// TIA Portal project "HEAT-1-CADIZ-S71500_V9" (V20)

(* hardware
DEVICE "S7-1500/ET200MP station_1"  S7-1500 station
   slot 0: "Rail_0"  Rack  6ES7 590-1***0-0AA0
   slot 1: "PLC_1"  CPU 1517F-3 PN/DP  6ES7 517-3FP00-0AB0  V3.0
      slot 3: "CPU display_1"  6ES7591-1BA00-0AA0
      slot 32768: "PROFINET interface_1"  X1
         slot 32769: "Port_1"  X1 P1
         slot 32770: "Port_2"  X1 P2
      slot 33024: "PROFINET interface_2"  X2
         slot 33025: "Port_1"  X2 P1
      slot 33280: "DP interface_1"  X3
      slot 34817: "Virtual CP interface port_1"  Virtual CP interface port  Virtual CP interface port
DEVICE "GSD device_1"  GSD.Device.PN
   slot 0: "Rack"  Rack  V1.0
   slot 0: "KRC5"  KUKA.PROFINET 6.0  0x300  V6.0
      slot 0: "KUKA.PROFINET 6.0"  KUKA.PROFINET 6.0
      slot 1: "Interface1"  Interface1
         slot 1: "Port001(XF3)"  Port001(XF3)
         slot 2: "Port002(XF4)"  Port002(XF4)
         slot 3: "Port003(XF5)"  Port003(XF5)
         slot 4: "Port004(XF6)"  Port004(XF6)
   slot 1: "64 safe digital in- and outputs (2.4)_1"  64 safe digital in- and outputs (2.4)  KUKADevF64_2.4
      slot 0: "64 safe digital in- and outputs (2.4)"  64 safe digital in- and outputs (2.4)
   slot 2: "256 digital in- and outputs_1"  256 digital in- and outputs  KUKA Device IO256
      slot 0: "256 digital in- and outputs"  256 digital in- and outputs
DEVICE "ET 200SP station_2"  ET 200SP-Station
   slot 0: "Rack_0"  Rack  6ES5 710-8MAx1
   slot 0: "islaparking"  IM 155-6 PN ST  6ES7 155-6AU01-0BN0  V4.2
   slot 1: "DI 16x24VDC ST_1"  DI 16x24VDC ST  6ES7 131-6BH01-0BA0  V0.0
      slot 1: "DI 16x24VDC ST_1"  DI 16x24VDC ST
   slot 2: "DI 8x24VDC ST_1"  DI 8x24VDC ST  6ES7 131-6BF01-0BA0  V0.0
      slot 1: "DI 8x24VDC ST_1"  DI 8x24VDC ST
   slot 3: "DQ 16x24VDC/0.5A ST_1"  DQ 16x24VDC/0.5A ST  6ES7 132-6BH01-0BA0  V0.0
      slot 1: "DQ 16x24VDC/0.5A ST_1"  DQ 16x24VDC/0.5A ST
   slot 4: "DQ 8x24VDC/0.5A ST_1"  DQ 8x24VDC/0.5A ST  6ES7 132-6BF01-0BA0  V0.0
      slot 1: "DQ 8x24VDC/0.5A ST_1"  DQ 8x24VDC/0.5A ST
   slot 5: "Server module_1"  Server module  6ES7 193-6PA00-0AA0  V1.1
      slot 1: "Server module_1"  Server module
   slot 127: "BA 2xRJ45"  BA 2xRJ45  6ES7 193-6AR00-0AA0  V0.0
      slot 1: "Port_1"  X1 P1R  6ES7 193-6AR00-0AA0  V0.0
      slot 2: "Port_2"  X1 P2R  6ES7 193-6AR00-0AA0  V0.0
DEVICE "ET 200SP station_1"  ET 200SP-Station
   slot 0: "Rack_0"  Rack  6ES5 710-8MAx1
   slot 0: "islarobot"  IM 155-6 PN ST  6ES7 155-6AU01-0BN0  V4.2
   slot 1: "DI 16x24VDC ST_1"  DI 16x24VDC ST  6ES7 131-6BH01-0BA0  V0.0
      slot 1: "DI 16x24VDC ST_1"  DI 16x24VDC ST
   slot 2: "DI 8x24VDC ST_1"  DI 8x24VDC ST  6ES7 131-6BF01-0BA0  V0.0
      slot 1: "DI 8x24VDC ST_1"  DI 8x24VDC ST
   slot 3: "DQ 16x24VDC/0.5A ST_1"  DQ 16x24VDC/0.5A ST  6ES7 132-6BH01-0BA0  V0.0
      slot 1: "DQ 16x24VDC/0.5A ST_1"  DQ 16x24VDC/0.5A ST
   slot 4: "DQ 8x24VDC/0.5A ST_1"  DQ 8x24VDC/0.5A ST  6ES7 132-6BF01-0BA0  V0.0
      slot 1: "DQ 8x24VDC/0.5A ST_1"  DQ 8x24VDC/0.5A ST
   slot 5: "Server module_1"  Server module  6ES7 193-6PA00-0AA0  V1.1
      slot 1: "Server module_1"  Server module
   slot 127: "BA 2xRJ45"  BA 2xRJ45  6ES7 193-6AR00-0AA0  V0.0
      slot 1: "Port_1"  X1 P1R  6ES7 193-6AR00-0AA0  V0.0
      slot 2: "Port_2"  X1 P2R  6ES7 193-6AR00-0AA0  V0.0
*)

// ===== PLC "PLC_1"  CPU 1517F-3 PN/DP =====

VAR_GLOBAL   // PLC tag table "Default tag table"
   "RES1 (reservado)" AT %Q500.0 : Bool;
   "eStopButtonCabinet" AT %I40.0 : Bool;   // Emergency-Stop cabinet — 1oo2 result
   "eStopButtonTank" AT %I40.1 : Bool;   // Emergency-Stop tank — 1oo2 result
   "eStopButtonTankPartnerCh" AT %I41.1 : Bool;   // partner channel 1oo2 — do not use
   "eStopButtonWaterSystem" AT %I40.2 : Bool;   // Emergency-Stop water system — 1oo2 result
   "eStopButtonWaterSystemPartnerCh" AT %I41.2 : Bool;   // partner channel 1oo2 — do not use
   "eStopButtonHmiPanel" AT %I40.3 : Bool;   // Emergency-Stop HMI panel — 1oo2 result
   "eStopButtonHmiPanelPartnerCh" AT %I41.3 : Bool;   // partner channel 1oo2 — do not use
   "eStopButtonLightCurtain1" AT %I40.4 : Bool;   // Emergency-Stop light curtain 1 — 1oo2 resul
   "eStopButtonLightCurtain1PartnerCh" AT %I41.4 : Bool;   // partner channel 1oo2 — do not use
   "eStopButtonDoor" AT %I40.5 : Bool;   // Emergency-Stop Door — 1oo2 result
   "eStopButtonDoorPartnerCh" AT %I41.5 : Bool;   // partner channel 1oo2 — do not use
   "lightCurtain1Ossd1" AT %I50.0 : Bool;   // Z2 – LC 1 OSSD 1 (receiver)
   "lightCurtain1Ossd2" AT %I51.0 : Bool;   // Z2 – LC 1 OSSD 2 (receiver)
   "lightCurtain3Ossd1" AT %I50.1 : Bool;   // Z2 – LC 3 OSSD 1 (receiver)
   "lightCurtain3Ossd2" AT %I51.1 : Bool;   // Z2 – LC 3 OSSD 2 (receiver)
   "lightCurtain6Ossd1" AT %I50.2 : Bool;   // Z2 – LC 6 OSSD 1 (receiver)
   "lightCurtain6Ossd2" AT %I51.2 : Bool;   // Z2 – LC 6 OSSD 2 (receiver)
   "enableAccessReqSelector" AT %I50.3 : Bool;   // Rotary selector – enabless request access
   "DoorClosedCh1" AT %I50.6 : Bool;   // Safety door closed interlock – contact 1
   "resetDoorButton" AT %I50.7 : Bool;   // Reset push‑button
   "SAF_DOOR_CLSD_CH2" AT %I51.6 : Bool;   // Safety door closed interlock – contact 2
   "SAF_DOOR_UNLOCK_CH1" AT %Q60.0 : Bool;   // Unlock safety door – redundant output 1
   "SAF_GATE_UNLOCK_CH2" AT %Q60.2 : Bool;   // Unlock safety door – redundant output 2
   "IND_RESET_LAMP" AT %Q10.0 : Bool;   // Reset indicator lamp
   "IND_STATUS_LAMP" AT %Q10.1 : Bool;   // System-status pilot light
   "CMD_PRESS_EXH_VALVE" AT %Q11.0 : Bool;   // Pressure/exhaust solenoid-valve command
   "STS_RECIRC_PUMP" AT %I20.0 : Bool;   // Recirculation-pump feedback
   "STS_TRANSFER_PUMP" AT %I20.1 : Bool;   // Transfer-pump feedback
   "ALM_UV_FILTER" AT %I20.2 : Bool;   // UV-filter fault alarm
   "ALM_PIT_LVL_LOW" AT %I20.3 : Bool;   // Sump low-level alarm
   "ALM_TANK_LVL_LOW" AT %I20.4 : Bool;   // Tank low-level alarm
   "STS_TANK_FILLING" AT %I20.5 : Bool;   // Tank filling status
   "STS_TANK_DRAINING" AT %I20.6 : Bool;   // Tank draining status
   "CMD_TANK_FILL" AT %Q30.0 : Bool;   // Fill tank command
   "CMD_TANK_DRAIN" AT %Q30.1 : Bool;   // Drain tank command
   "MODE_WATER_MAN" AT %Q30.2 : Bool;   // Water system manual mode
   "MODE_WATER_AUTO" AT %Q30.3 : Bool;   // Water system automatic mode
   "IND_BEACON2_GREEN" AT %Q30.4 : Bool;   // Beacon 2 – green
   "IND_BEACON2_RED" AT %Q30.5 : Bool;   // Beacon 2 – red
   "robotPresenceSignalZone1" AT %I500.0 : Bool;
   "robotPresenceSignalZone2" AT %I500.1 : Bool;
   "robotPresenceSignalZone3" AT %I500.2 : Bool;
   "eStopButtonCabinetPartnerCh" AT %I41.0 : Bool;   // partner channel 1oo2 — do not use
   "lightCurtain2Ossd1" AT %I300.0 : Bool;
   "lightCurtain2Ossd2" AT %I301.0 : Bool;
   "eStopButtonIslandRightPartner" AT %I301.1 : Bool;
   "lightCurtain4Ossd1" AT %I350.0 : Bool;
   "eStopButtonIslandLeft" AT %I350.1 : Bool;
   "lightCurtain5Ossd1" AT %I350.2 : Bool;
   "eStopButtonIslandLefttPartner" AT %I350.3 : Bool;   // partner channel 1oo2 — do not use
   "lightCurtain4Ossd2" AT %I350.4 : Bool;
   "lightCurtain5Ossd2" AT %I350.6 : Bool;
   "accessReqButtonZone2" AT %I51.4 : Bool;   // Illuminated push-button – access request for zone 2
   "accessReqButtonZone3" AT %I51.5 : Bool;   // Illuminated push-button – access request for zone 3
   "accessReqButtonZone1" AT %I51.3 : Bool;   // Illuminated push-button – access request for zone 1
   "eStopButtonIslandRight" AT %I300.1 : Bool;
   "NHE – E‑Stop externo  NO pulsado" AT %Q500.1 : Bool;
   "BS – Puerta cerrada" AT %Q500.2 : Bool;
   "QBS – Ack puerta" AT %Q500.3 : Bool;
   "SHS1 – Stop 1" AT %Q500.4 : Bool;
   "SHS2 – Stop 2" AT %Q500.5 : Bool;
   "RES6" AT %Q500.6 : Bool;
   "RES7" AT %Q500.7 : Bool;
   "US2 – 24 V US2" AT %Q501.0 : Bool;
   "SBH – Safe Op Stop" AT %Q501.1 : Bool;
   "RES11" AT %Q501.2 : Bool;
   "RES12" AT %Q501.3 : Bool;
   "RES13" AT %Q501.4 : Bool;
   "RES14" AT %Q501.5 : Bool;
   "RES15" AT %Q501.6 : Bool;
   "SPA – Power‑down Ack" AT %Q501.7 : Bool;
   "resetHmiButton" AT %I51.7 : Bool;
   "Tag_1" AT %M200.0 : Bool;
   "Tag_2" AT %M201.0 : Bool;
   "Tag_3" AT %M500.1 : Bool;
   "Tag_4" AT %M755.5 : Bool;
   "Tag_5" AT %QB600 : Byte;
   "V5" AT %Q0.4 : Bool;
   "ABRIR_TAPA_PEPA" AT %Q170.2 : Bool;
   "CERRAR_TAPA_PEPA" AT %Q170.3 : Bool;
   "ABRIR_TAPA_INMERSION" AT %Q170.4 : Bool;
   "CERRAR_TAPA_INMERSION" AT %Q170.5 : Bool;
   "ABRIR_TAPA_MARCADOR" AT %Q170.6 : Bool;
   "CERRAR_TAPA_MARCADOR" AT %Q170.7 : Bool;
   "ABRIR_TAPA_PERFILOMETRO" AT %Q171.0 : Bool;
   "CERRAR_TAPA_PERFILOMETRO" AT %Q171.1 : Bool;
   "V6" AT %Q0.5 : Bool;
   "V7" AT %Q0.6 : Bool;
   "V8" AT %Q0.7 : Bool;
END_VAR

VAR_GLOBAL   // PLC tag table "Robot Jog"
   "tcpTargetX_01" AT %Q600.1 : Bool;
   "tcpTargetX_02" AT %Q600.2 : Bool;
   "tcpTargetX_03" AT %Q600.3 : Bool;
   "tcpTargetX_04" AT %Q600.4 : Bool;
   "tcpTargetX_05" AT %Q600.5 : Bool;
   "tcpTargetX_08" AT %Q601.0 : Bool;
   "tcpTargetX_16" AT %Q602.0 : Bool;
   "tcpTargetX_17" AT %Q602.1 : Bool;
   "tcpTargetX_06" AT %Q600.6 : Bool;
   "tcpTargetX_07" AT %Q600.7 : Bool;
   "tcpTargetX_09" AT %Q601.1 : Bool;
   "tcpTargetX_10" AT %Q601.2 : Bool;
   "tcpTargetX_11" AT %Q601.3 : Bool;
   "tcpTargetX_12" AT %Q601.4 : Bool;
   "tcpTargetX_13" AT %Q601.5 : Bool;
   "tcpTargetX_14" AT %Q601.6 : Bool;
   "tcpTargetX_15" AT %Q601.7 : Bool;
   "tcpTargetX_18" AT %Q602.2 : Bool;
   "tcpTargetX_19" AT %Q602.3 : Bool;
   "tcpTargetX_20" AT %Q602.4 : Bool;
   "tcpTargetX_21" AT %Q602.5 : Bool;
   "tcpTargetX_22" AT %Q602.6 : Bool;
   "tcpTargetX_23" AT %Q602.7 : Bool;
   "tcpTargetX_24" AT %Q603.0 : Bool;
   "tcpTargetX_25" AT %Q603.1 : Bool;
   "tcpTargetX_26" AT %Q603.2 : Bool;
   "tcpTargetX_27" AT %Q603.3 : Bool;
   "tcpTargetX_28" AT %Q603.4 : Bool;
   "tcpTargetX_29" AT %Q603.5 : Bool;
   "tcpTargetX_30" AT %Q603.6 : Bool;
   "tcpTargetX_31" AT %Q603.7 : Bool;
   "tcpTargetY_00" AT %Q604.0 : Bool;
   "tcpTargetY_01" AT %Q604.1 : Bool;
   "tcpTargetY_02" AT %Q604.2 : Bool;
   "tcpTargetY_03" AT %Q604.3 : Bool;
   "tcpTargetY_04" AT %Q604.4 : Bool;
   "tcpTargetY_05" AT %Q604.5 : Bool;
   "tcpTargetY_06" AT %Q604.6 : Bool;
   "tcpTargetY_07" AT %Q604.7 : Bool;
   "tcpTargetY_08" AT %Q605.0 : Bool;
   "tcpTargetY_09" AT %Q605.1 : Bool;
   "tcpTargetY_10" AT %Q605.2 : Bool;
   "tcpTargetY_11" AT %Q605.3 : Bool;
   "tcpTargetY_12" AT %Q605.4 : Bool;
   "tcpTargetY_13" AT %Q605.5 : Bool;
   "tcpTargetY_14" AT %Q605.6 : Bool;
   "tcpTargetY_15" AT %Q605.7 : Bool;
   "tcpTargetY_16" AT %Q606.0 : Bool;   // $IN[49]
   "tcpTargetY_17" AT %Q606.1 : Bool;   // $IN[50]
   "tcpTargetY_18" AT %Q606.2 : Bool;   // $IN[51]
   "tcpTargetY_19" AT %Q606.3 : Bool;   // true
   "tcpTargetY_20" AT %Q606.4 : Bool;
   "tcpTargetY_21" AT %Q606.5 : Bool;   // true
   "tcpTargetY_22" AT %Q606.6 : Bool;   // true
   "tcpTargetY_23" AT %Q606.7 : Bool;   // true
   "tcpTargetY_24" AT %Q607.0 : Bool;   // true
   "tcpTargetY_25" AT %Q607.1 : Bool;   // true
   "tcpTargetY_26" AT %Q607.2 : Bool;   // true
   "tcpTargetY_27" AT %Q607.3 : Bool;
   "tcpTargetY_28" AT %Q607.4 : Bool;
   "tcpTargetY_29" AT %Q607.5 : Bool;
   "tcpTargetY_30" AT %Q607.6 : Bool;
   "tcpTargetY_31" AT %Q607.7 : Bool;
   "tcpTargetZ_00" AT %Q608.0 : Bool;
   "tcpTargetZ_01" AT %Q608.1 : Bool;
   "tcpTargetZ_02" AT %Q608.2 : Bool;
   "tcpTargetZ_03" AT %Q608.3 : Bool;
   "tcpTargetZ_04" AT %Q608.4 : Bool;
   "tcpTargetZ_05" AT %Q608.5 : Bool;
   "tcpTargetZ_06" AT %Q608.6 : Bool;
   "tcpTargetZ_07" AT %Q608.7 : Bool;
   "tcpTargetZ_08" AT %Q609.0 : Bool;
   "tcpTargetZ_09" AT %Q609.1 : Bool;
   "tcpTargetZ_10" AT %Q609.2 : Bool;
   "tcpTargetZ_11" AT %Q609.3 : Bool;
   "tcpTargetZ_12" AT %Q609.4 : Bool;
   "tcpTargetZ_13" AT %Q609.5 : Bool;
   "tcpTargetZ_14" AT %Q609.6 : Bool;
   "tcpTargetZ_15" AT %Q609.7 : Bool;
   "tcpTargetZ_16" AT %Q610.0 : Bool;
   "tcpTargetZ_17" AT %Q610.1 : Bool;
   "tcpTargetZ_18" AT %Q610.2 : Bool;
   "tcpTargetZ_19" AT %Q610.3 : Bool;
   "tcpTargetZ_20" AT %Q610.4 : Bool;
   "tcpTargetZ_21" AT %Q610.5 : Bool;
   "tcpTargetZ_22" AT %Q610.6 : Bool;
   "tcpTargetZ_23" AT %Q610.7 : Bool;
   "tcpTargetZ_24" AT %Q611.0 : Bool;
   "tcpTargetZ_25" AT %Q611.1 : Bool;
   "tcpTargetZ_26" AT %Q611.2 : Bool;
   "tcpTargetZ_27" AT %Q611.3 : Bool;
   "tcpTargetZ_28" AT %Q611.4 : Bool;
   "tcpTargetZ_29" AT %Q611.5 : Bool;
   "tcpTargetZ_30" AT %Q611.6 : Bool;
   "tcpTargetZ_31" AT %Q611.7 : Bool;
   "e1Target_00" AT %Q612.0 : Bool;
   "e1Target_01" AT %Q612.1 : Bool;
   "e1Target_02" AT %Q612.2 : Bool;
   "e1Target_03" AT %Q612.3 : Bool;
   "e1Target_04" AT %Q612.4 : Bool;
   "e1Target_05" AT %Q612.5 : Bool;
   "e1Target_06" AT %Q612.6 : Bool;
   "e1Target_07" AT %Q612.7 : Bool;
   "e1Target_08" AT %Q613.0 : Bool;
   "e1Target_09" AT %Q613.1 : Bool;
   "e1Target_10" AT %Q613.2 : Bool;
   "e1Target_11" AT %Q613.3 : Bool;
   "e1Target_12" AT %Q613.4 : Bool;
   "e1Target_13" AT %Q613.5 : Bool;
   "e1Target_14" AT %Q613.6 : Bool;
   "e1Target_15" AT %Q613.7 : Bool;
   "e1Target_16" AT %Q614.0 : Bool;
   "e1Target_17" AT %Q614.1 : Bool;
   "e1Target_18" AT %Q614.2 : Bool;
   "e1Target_19" AT %Q614.3 : Bool;
   "e1Target_20" AT %Q614.4 : Bool;
   "e1Target_21" AT %Q614.5 : Bool;
   "e1Target_22" AT %Q614.6 : Bool;
   "e1Target_23" AT %Q614.7 : Bool;
   "e1Target_24" AT %Q615.0 : Bool;
   "e1Target_25" AT %Q615.1 : Bool;
   "e1Target_26" AT %Q615.2 : Bool;
   "e1Target_27" AT %Q615.3 : Bool;
   "e1Target_28" AT %Q615.4 : Bool;
   "e1Target_29" AT %Q615.5 : Bool;
   "e1Target_30" AT %Q615.6 : Bool;
   "e1Target_31" AT %Q615.7 : Bool;
   "e1Target_Word" AT %QD612 : DWord;
   "moveCodeKuka" AT %QW616 : Word;   // SIGNAL goTrrigger $IN[ 129]
   "rbDone" AT %I624.0 : Bool;   // SIGNAL rbDoneEdge $OUT[193]
   "x1Target_Word" AT %QD600 : DWord;
   "y1Target_Word" AT %QD604 : DWord;
   "z1Target_Word" AT %QD608 : DWord;
   "goTrigger" AT %Q618.0 : Bool;
END_VAR

VAR_GLOBAL   // PLC tag table "Robot Position"
   "tcpPosX_00" AT %I600.0 : Bool;
   "tcpPosX_01" AT %I600.1 : Bool;
   "tcpPosX_02" AT %I600.2 : Bool;
   "tcpPosX_03" AT %I600.3 : Bool;
   "tcpPosX_04" AT %I600.4 : Bool;
   "tcpPosX_05" AT %I600.5 : Bool;
   "tcpPosX_06" AT %I600.6 : Bool;
   "tcpPosX_07" AT %I600.7 : Bool;
   "tcpPosX_08" AT %I601.0 : Bool;
   "tcpPosX_09" AT %I601.1 : Bool;
   "tcpPosX_10" AT %I601.2 : Bool;
   "tcpPosX_11" AT %I601.3 : Bool;
   "tcpPosX_12" AT %I601.4 : Bool;
   "tcpPosX_13" AT %I601.5 : Bool;
   "tcpPosX_14" AT %I601.6 : Bool;
   "tcpPosX_15" AT %I601.7 : Bool;
   "tcpPosX_16" AT %I602.0 : Bool;
   "tcpPosX_17" AT %I602.1 : Bool;
   "tcpPosX_18" AT %I602.2 : Bool;
   "tcpPosX_19" AT %I602.3 : Bool;
   "tcpPosX_20" AT %I602.4 : Bool;
   "tcpPosX_21" AT %I602.5 : Bool;
   "tcpPosX_22" AT %I602.6 : Bool;
   "tcpPosX_23" AT %I602.7 : Bool;
   "tcpPosX_24" AT %I603.0 : Bool;
   "tcpPosX_25" AT %I603.1 : Bool;
   "tcpPosX_26" AT %I603.2 : Bool;
   "tcpPosX_27" AT %I603.3 : Bool;
   "tcpPosX_28" AT %I603.4 : Bool;
   "tcpPosX_29" AT %I603.5 : Bool;
   "tcpPosX_30" AT %I603.6 : Bool;
   "tcpPosX_31" AT %I603.7 : Bool;
   "tcpPosY_00" AT %I604.0 : Bool;
   "tcpPosY_01" AT %I604.1 : Bool;
   "tcpPosY_02" AT %I604.2 : Bool;
   "tcpPosY_03" AT %I604.3 : Bool;
   "tcpPosY_04" AT %I604.4 : Bool;
   "tcpPosY_05" AT %I604.5 : Bool;
   "tcpPosY_06" AT %I604.6 : Bool;
   "tcpPosY_07" AT %I604.7 : Bool;
   "tcpPosY_08" AT %I605.0 : Bool;
   "tcpPosY_09" AT %I605.1 : Bool;
   "tcpPosY_10" AT %I605.2 : Bool;
   "tcpPosY_11" AT %I605.3 : Bool;
   "tcpPosY_12" AT %I605.4 : Bool;
   "tcpPosY_13" AT %I605.5 : Bool;
   "tcpPosY_14" AT %I605.6 : Bool;
   "tcpPosY_15" AT %I605.7 : Bool;
   "tcpPosY_16" AT %I606.0 : Bool;
   "tcpPosY_17" AT %I606.1 : Bool;
   "tcpPosY_18" AT %I606.2 : Bool;
   "tcpPosY_19" AT %I606.3 : Bool;
   "tcpPosY_20" AT %I606.4 : Bool;
   "tcpPosY_21" AT %I606.5 : Bool;
   "tcpPosY_22" AT %I606.6 : Bool;
   "tcpPosY_23" AT %I606.7 : Bool;
   "tcpPosY_24" AT %I607.0 : Bool;
   "tcpPosY_25" AT %I607.1 : Bool;
   "tcpPosY_26" AT %I607.2 : Bool;
   "tcpPosY_27" AT %I607.3 : Bool;
   "tcpPosY_28" AT %I607.4 : Bool;
   "tcpPosY_29" AT %I607.5 : Bool;
   "tcpPosY_30" AT %I607.6 : Bool;
   "tcpPosY_31" AT %I607.7 : Bool;
   "tcpPosZ_00" AT %I608.0 : Bool;
   "tcpPosZ_01" AT %I608.1 : Bool;
   "tcpPosZ_02" AT %I608.2 : Bool;
   "tcpPosZ_03" AT %I608.3 : Bool;
   "tcpPosZ_04" AT %I608.4 : Bool;
   "tcpPosZ_05" AT %I608.5 : Bool;
   "tcpPosZ_06" AT %I608.6 : Bool;
   "tcpPosZ_07" AT %I608.7 : Bool;
   "tcpPosZ_08" AT %I609.0 : Bool;
   "tcpPosZ_09" AT %I609.1 : Bool;
   "tcpPosZ_10" AT %I609.2 : Bool;
   "tcpPosZ_11" AT %I609.3 : Bool;
   "tcpPosZ_12" AT %I609.4 : Bool;
   "tcpPosZ_13" AT %I609.5 : Bool;
   "tcpPosZ_14" AT %I609.6 : Bool;
   "tcpPosZ_15" AT %I609.7 : Bool;
   "tcpPosZ_16" AT %I610.0 : Bool;
   "tcpPosZ_17" AT %I610.1 : Bool;
   "tcpPosZ_18" AT %I610.2 : Bool;
   "tcpPosZ_19" AT %I610.3 : Bool;
   "tcpPosZ_20" AT %I610.4 : Bool;
   "tcpPosZ_21" AT %I610.5 : Bool;
   "tcpPosZ_22" AT %I610.6 : Bool;
   "tcpPosZ_23" AT %I610.7 : Bool;
   "tcpPosZ_24" AT %I611.0 : Bool;
   "tcpPosZ_25" AT %I611.1 : Bool;
   "tcpPosZ_26" AT %I611.2 : Bool;
   "tcpPosZ_27" AT %I611.3 : Bool;
   "tcpPosZ_28" AT %I611.4 : Bool;
   "tcpPosZ_29" AT %I611.5 : Bool;
   "tcpPosZ_30" AT %I611.6 : Bool;
   "tcpPosZ_31" AT %I611.7 : Bool;
   "tcpPosA_00" AT %I612.0 : Bool;
   "tcpPosA_01" AT %I612.1 : Bool;
   "tcpPosA_02" AT %I612.2 : Bool;
   "tcpPosA_03" AT %I612.3 : Bool;
   "tcpPosA_04" AT %I612.4 : Bool;
   "tcpPosA_05" AT %I612.5 : Bool;
   "tcpPosA_06" AT %I612.6 : Bool;
   "tcpPosA_07" AT %I612.7 : Bool;
   "tcpPosA_08" AT %I613.0 : Bool;
   "tcpPosA_09" AT %I613.1 : Bool;
   "tcpPosA_10" AT %I613.2 : Bool;
   "tcpPosA_11" AT %I613.3 : Bool;
   "tcpPosA_12" AT %I613.4 : Bool;
   "tcpPosA_13" AT %I613.5 : Bool;
   "tcpPosA_14" AT %I613.6 : Bool;
   "tcpPosA_15" AT %I613.7 : Bool;
   "tcpPosA_16" AT %I614.0 : Bool;
   "tcpPosA_17" AT %I614.1 : Bool;
   "tcpPosA_18" AT %I614.2 : Bool;
   "tcpPosA_19" AT %I614.3 : Bool;
   "tcpPosA_20" AT %I614.4 : Bool;
   "tcpPosA_21" AT %I614.5 : Bool;
   "tcpPosA_22" AT %I614.6 : Bool;
   "tcpPosA_23" AT %I614.7 : Bool;
   "tcpPosA_24" AT %I615.0 : Bool;
   "tcpPosA_25" AT %I615.1 : Bool;
   "tcpPosA_26" AT %I615.2 : Bool;
   "tcpPosA_27" AT %I615.3 : Bool;
   "tcpPosA_28" AT %I615.4 : Bool;
   "tcpPosA_29" AT %I615.5 : Bool;
   "tcpPosA_30" AT %I615.6 : Bool;
   "tcpPosA_31" AT %I615.7 : Bool;
   "tcpPosB_00" AT %I616.0 : Bool;
   "tcpPosB_01" AT %I616.1 : Bool;
   "tcpPosB_02" AT %I616.2 : Bool;
   "tcpPosB_03" AT %I616.3 : Bool;
   "tcpPosB_04" AT %I616.4 : Bool;
   "tcpPosB_05" AT %I616.5 : Bool;
   "tcpPosB_06" AT %I616.6 : Bool;
   "tcpPosB_07" AT %I616.7 : Bool;
   "tcpPosB_08" AT %I617.0 : Bool;
   "tcpPosB_09" AT %I617.1 : Bool;
   "tcpPosB_10" AT %I617.2 : Bool;
   "tcpPosB_11" AT %I617.3 : Bool;
   "tcpPosB_12" AT %I617.4 : Bool;
   "tcpPosB_13" AT %I617.5 : Bool;
   "tcpPosB_14" AT %I617.6 : Bool;
   "tcpPosB_15" AT %I617.7 : Bool;
   "tcpPosB_16" AT %I618.0 : Bool;
   "tcpPosB_17" AT %I618.1 : Bool;
   "tcpPosB_18" AT %I618.2 : Bool;
   "tcpPosB_19" AT %I618.3 : Bool;
   "tcpPosB_20" AT %I618.4 : Bool;
   "tcpPosB_21" AT %I618.5 : Bool;
   "tcpPosB_22" AT %I618.6 : Bool;
   "tcpPosB_23" AT %I618.7 : Bool;
   "tcpPosB_24" AT %I619.0 : Bool;
   "tcpPosB_25" AT %I619.1 : Bool;
   "tcpPosB_26" AT %I619.2 : Bool;
   "tcpPosB_27" AT %I619.3 : Bool;
   "tcpPosB_28" AT %I619.4 : Bool;
   "tcpPosB_29" AT %I619.5 : Bool;
   "tcpPosB_30" AT %I619.6 : Bool;
   "tcpPosB_31" AT %I619.7 : Bool;
   "tcpPosC_00" AT %I620.0 : Bool;
   "tcpPosC_01" AT %I620.1 : Bool;
   "tcpPosC_02" AT %I620.2 : Bool;
   "tcpPosC_03" AT %I620.3 : Bool;
   "tcpPosC_04" AT %I620.4 : Bool;
   "tcpPosC_05" AT %I620.5 : Bool;
   "tcpPosC_06" AT %I620.6 : Bool;
   "tcpPosC_07" AT %I620.7 : Bool;
   "tcpPosC_08" AT %I621.0 : Bool;
   "tcpPosC_09" AT %I621.1 : Bool;
   "tcpPosC_10" AT %I621.2 : Bool;
   "tcpPosC_11" AT %I621.3 : Bool;
   "tcpPosC_12" AT %I621.4 : Bool;
   "tcpPosC_13" AT %I621.5 : Bool;
   "tcpPosC_14" AT %I621.6 : Bool;
   "tcpPosC_15" AT %I621.7 : Bool;
   "tcpPosC_16" AT %I622.0 : Bool;
   "tcpPosC_17" AT %I622.1 : Bool;
   "tcpPosC_18" AT %I622.2 : Bool;
   "tcpPosC_19" AT %I622.3 : Bool;
   "tcpPosC_20" AT %I622.4 : Bool;
   "tcpPosC_21" AT %I622.5 : Bool;
   "tcpPosC_22" AT %I622.6 : Bool;
   "tcpPosC_23" AT %I622.7 : Bool;
   "tcpPosC_24" AT %I623.0 : Bool;
   "tcpPosC_25" AT %I623.1 : Bool;
   "tcpPosC_26" AT %I623.2 : Bool;
   "tcpPosC_27" AT %I623.3 : Bool;
   "tcpPosC_28" AT %I623.4 : Bool;
   "tcpPosC_29" AT %I623.5 : Bool;
   "tcpPosC_30" AT %I623.6 : Bool;
   "tcpPosC_31" AT %I623.7 : Bool;
   "tcpPosE1_01" AT %I628.0 : Bool;
   "tcpPosE1_02" AT %I628.1 : Bool;
   "tcpPosE1_03" AT %I628.2 : Bool;
   "tcpPosE1_04" AT %I628.3 : Bool;
   "tcpPosE1_05" AT %I628.4 : Bool;
   "tcpPosE1_06" AT %I628.5 : Bool;
   "tcpPosE1_07" AT %I628.6 : Bool;
   "tcpPosE1_08" AT %I628.7 : Bool;
   "tcpPosE1_09" AT %I629.0 : Bool;
   "tcpPosE1_10" AT %I629.1 : Bool;
   "tcpPosE1_11" AT %I629.2 : Bool;
   "tcpPosE1_12" AT %I629.3 : Bool;
   "tcpPosE1_13" AT %I629.4 : Bool;
   "tcpPosE1_14" AT %I629.5 : Bool;
   "tcpPosE1_15" AT %I629.6 : Bool;
   "tcpPosE1_16" AT %I629.7 : Bool;
   "tcpPosE1_17" AT %I630.0 : Bool;
   "tcpPosE1_18" AT %I630.1 : Bool;
   "tcpPosE1_19" AT %I630.2 : Bool;
   "tcpPosE1_20" AT %I630.3 : Bool;
   "tcpPosE1_21" AT %I630.4 : Bool;
   "tcpPosE1_22" AT %I630.5 : Bool;
   "tcpPosE1_23" AT %I630.6 : Bool;
   "tcpPosE1_24" AT %I630.7 : Bool;
   "tcpPosE1_25" AT %I631.0 : Bool;
   "tcpPosE1_26" AT %I631.1 : Bool;
   "tcpPosE1_27" AT %I631.2 : Bool;
   "tcpPosE1_28" AT %I631.3 : Bool;
   "tcpPosE1_29" AT %I631.4 : Bool;
   "tcpPosE1_30" AT %I631.5 : Bool;
   "tcpPosE1_31" AT %I631.6 : Bool;
   "tcpPosE1_32" AT %I631.7 : Bool;
   "tcpX_rawLe32" AT %ID600 : DWord;
   "tcpY_rawLe32" AT %ID604 : DWord;
   "tcpZ_rawLe32" AT %ID608 : DWord;
   "tcpB_rawLe32" AT %ID616 : DWord;
   "tcpC_rawLe32" AT %ID620 : DWord;
   "e1_rawLe32" AT %ID628 : DWord;
   "tcpA_rawLe32" AT %ID612 : DWord;
END_VAR

VAR_GLOBAL   // PLC tag table "Tool Change"
   "dockSensorToolInPosition" AT %I150.0 : Bool;   // DETECTOR_YUGO_LP
   "dockSensorCoverClosed" AT %I150.1 : Bool;   // TAPA_CERRADA_YUGO_LP
   "dockSensorCoverOpen" AT %I160.0 : Bool;   // TAPA_ABIERTA_YUGO_LP
   "dockValveV2UnlockOn" AT %Q171.2 : Bool;   // SOLTAR_HERRAMIENTA_YUGO_LP / CAMBIA A FALSE
   "dockValveCoverOpenOn" AT %Q170.0 : Bool;   // ABRIR_TAPA_YUGO_LP
   "dockValveCoverCloseOn" AT %Q170.1 : Bool;   // CERRAR_TAPA_YUGO_LP
   "robotSensorMpsUnlocked" AT %I200.0 : Bool;   // INTERCAMBIO_DESBLOQUEADO_LR
   "robotSensorMpsLocked" AT %I200.1 : Bool;   // INTERCAMBIO_BLOQUEADO_LR
   "robotSensorMpsCoupled" AT %I200.2 : Bool;   // HERRAMIENTA_PUESTA_LR /AL COLOCAR METAL
   "robotSensorMpsCtrlAirPressureOk" AT %I200.3 : Bool;   // PRESION_CORRECTA_LR
   "kukaFeedbackDockToolInPosition" AT %Q618.1 : Bool;   // INKUKA_DETECTOR_HERRAMIENTA
   "kukaFeedbackDockCoverClosed" AT %Q618.2 : Bool;   // INKUKA_TAPA_CERRADA_YUGO
   "kukaFeedbackDockCoverOpen" AT %Q618.3 : Bool;   // INKUKA_TAPA_ABIERTA_YUGO
   "kukaFeedbackRobotMpsUnlocked" AT %Q618.4 : Bool;   // INKUKA_INTERCAMBIO_DESBLOQUEADO
   "kukaFeedbackRobotMpsLocked" AT %Q618.5 : Bool;   // INKUKA_INTERCAMBIO_BLOQUEADO
   "kukaFeedbackRobotMpsCoupled" AT %Q618.6 : Bool;   // INKUKA_HERRAMIENTA_PUESTA /AL COLOCAR util met
   "kukaFeedbackRobotMpsCtrlAirPressureOk" AT %Q618.7 : Bool;
   "kukaCmdUnlockMps" AT %I624.1 : Bool;   // OUTKUKA_SOLTAR_HERRAMIENTA_YUGO
   "kukaCmdOpenCover" AT %I624.2 : Bool;   // OUTKUKA_ABRIR_TAPA_YUGO
   "kukaCmdCloseCover" AT %I624.3 : Bool;   // OUTKUKA_CERRAR_TAPA_YUGO
   "V1_B14_S2" AT %Q0.0 : Bool;
   "V1_B12_S4" AT %Q0.1 : Bool;
   "V2_B14_S2" AT %Q0.2 : Bool;
   "V2_B12_S4" AT %Q0.3 : Bool;
END_VAR

// folder: 10. System/DbsInstancia

DATA_BLOCK "InstKukaControlSeq"   // DB14
{ S7_Optimized_Access := 'TRUE' }
VERSION : 0.1
// stored: InstanceOfName KukaControlSeq
"KukaControlSeq"
BEGIN
END_DATA_BLOCK

DATA_BLOCK "InstSupervisorSeq"   // DB15
{ S7_Optimized_Access := 'TRUE' }
VERSION : 0.1
// stored: InstanceOfName SupervisorSeq
"SupervisorSeq"
BEGIN
END_DATA_BLOCK

DATA_BLOCK "InstSeqManager"   // DB16
{ S7_Optimized_Access := 'TRUE' }
VERSION : 0.1
// stored: InstanceOfName SeqManager
"SeqManager"
BEGIN
END_DATA_BLOCK

// folder: 10. System/DbsOpcUa

DATA_BLOCK "PlcStatus"   // DB4
{ S7_Optimized_Access := 'TRUE' }
VERSION : 0.1
   VAR
      mode : Struct
         effective : UInt;
         ready : Bool;
      END_STRUCT;
      active : Struct
         baseId : UInt;
         toolId : UInt;
         profileId : UInt;
      END_STRUCT;
      exec : Struct
         ackSeq : UInt;
         accepted : Bool;
         busy : Bool;
         done : Bool;
         error : Bool;
         errorCode : UDInt;
      END_STRUCT;
      pose : Struct
         tcpPosX_mm : LReal;
         tcpPosY_mm : LReal;
         tcpPosZ_mm : LReal;
         tcpOriA_deg : LReal;
         tcpOriB_deg : LReal;
         tcpOriC_deg : LReal;
         e1Pos_mm : LReal;
      END_STRUCT;
      Supervisor : Struct
         global : Struct
            heartBeatPlc : Bool;
            stepPlc : Int;
            plcOk : Bool;
            safetyOk : Bool;
            airOk : Bool;
            inspWaterOk : Bool;
            tankWaterOk : Bool;
            robotOk : Bool;
            acknowledge : Bool;
         END_STRUCT;
         identification : Struct
            carriageId : UInt;
            newCarriageId : Bool;
            idRunning : Bool;
         END_STRUCT;
         startUs : Struct
            startUsReady : Bool;
         END_STRUCT;
         stopUs : Struct
            stopUsReady : Bool;
         END_STRUCT;
         "deadElementCheck&Balancing" : Struct
            paCheckReady : Bool;
         END_STRUCT;
         gaintAdjustment : Struct
            gainReady : Bool;
         END_STRUCT;
         "tcgCheck&Adj" : Struct
            tcgReady : Bool;
         END_STRUCT;
         scanGeneric : Struct
            idScan : String;
            pointOrigin : LReal;
            xSize : LReal;
            ySize : LReal;
         END_STRUCT;
         scanRefPart : Struct
            scanRefStart : Bool;
         END_STRUCT;
         scanInsPart : Struct
            scanInspStart : Bool;
         END_STRUCT;
         preEval : Struct
            markRunning : Bool;
            markState : Bool;
         END_STRUCT;
         "break/Unbreak" : Struct
            breakUs : Bool;
            unbreakUs : Bool;
         END_STRUCT;
         rescanning : Struct
            robotRescanning : Bool;
         END_STRUCT;
         error : Struct
            acknowledgeError : Bool;
         END_STRUCT;
      END_STRUCT;
   END_VAR
BEGIN
END_DATA_BLOCK

DATA_BLOCK "KukaControlCmd"   // DB5
{ S7_Optimized_Access := 'TRUE' }
VERSION : 0.1
   VAR
      code : UInt;
      seq : UInt;
      tcpTargetX_mm : LReal;
      tcpTargetY_mm : LReal;
      tcpTargetZ_mm : LReal;
      e1Target : LReal;
      toolRequestId : UInt;
      baseRequestId : UInt;
      profileRequestId : UInt;
      vel_mms : LReal;
      index_mm : LReal;
      apo_mm : LReal;
      mode : Struct
         request : UInt;
         reqSeq : UInt;
      END_STRUCT;
   END_VAR
BEGIN
END_DATA_BLOCK

DATA_BLOCK "SupervisorCmd"   // DB6
{ S7_Optimized_Access := 'TRUE' }
VERSION : 0.1
   VAR
      global : Struct
         heartBeatSupervisor : Bool;
         stepSupervisor : Int;
         supervisorOk : Bool;
         stateUs : Bool;
      END_STRUCT;
      request : Struct
         reqCarriageId : Bool;
         reqRefPart : Bool;
         reqStopCycle : Bool;
         reqTcgAdj : Bool;
         reqId : Bool;
         reqPreEval : Bool;
         reqIdentificationState : Bool;
         reqMark : Bool;
      END_STRUCT;
      identification : Struct
         pns : String;
         referencePart : String;
         endEffector : Int;
         utTech : UInt;
         teachReq : Bool;
         paCheckReq : Bool;
         tcgReq : Bool;
      END_STRUCT;
      startUs : Struct
         startUsRunning : Bool;
      END_STRUCT;
      stopUs : Struct
         stopUsRunning : Bool;
      END_STRUCT;
      "deadElementCheck&Balancing" : Struct
         elemState : Bool;
         elemRunning : Bool;
         balState : Bool;
         balRunning : Bool;
      END_STRUCT;
      gainAdjustment : Struct
         gainState : Bool;
         gainRunning : Bool;
      END_STRUCT;
      "tcgCheck&Adj" : Struct
         tcgInProgress : Bool;
         tcgNextStep : Bool;
         tcgState : Bool;
      END_STRUCT;
      scanRefPart : Struct
         scanRefState : Bool;
         scanRefRunning : Bool;
      END_STRUCT;
      scanInspPart : Struct
         scanInspState : Bool;
         scanInspRunning : Bool;
      END_STRUCT;
      preEval : Struct
         pointCoordinates : LReal;
      END_STRUCT;
      rescanning : Struct
         goBack : Bool;
         rescanning : Bool;
      END_STRUCT;
      error : Struct
         errorMessage : String;
         errorOcurred : Bool;
      END_STRUCT;
   END_VAR
BEGIN
END_DATA_BLOCK

// folder: 10. System/Utilities

DATA_BLOCK "ConstantsDB"   // DB37
{ S7_Optimized_Access := 'TRUE' }
VERSION : 0.1
BEGIN
END_DATA_BLOCK

// folder: 20. Robot Services/AutoExt

DATA_BLOCK "instAutoExtSeq"   // DB7
{ S7_Optimized_Access := 'TRUE' }
VERSION : 0.1
// stored: InstanceOfName AutoExtSeq
"AutoExtSeq"
BEGIN
END_DATA_BLOCK

// folder: 20. Robot Services/DbsInstancia

DATA_BLOCK "InstTcpJogging"   // DB2
{ S7_Optimized_Access := 'TRUE' }
VERSION : 0.1
// stored: InstanceOfName TcpJogging
"TcpJogging"
BEGIN
END_DATA_BLOCK

DATA_BLOCK "ToolChange_DB"   // DB8
{ S7_Optimized_Access := 'TRUE' }
VERSION : 0.1
// stored: InstanceOfName ToolChange
"ToolChange"
BEGIN
END_DATA_BLOCK

DATA_BLOCK "TcpPoseDecoderLe32_DB"   // DB10
{ S7_Optimized_Access := 'TRUE' }
VERSION : 0.1
// stored: InstanceOfName TcpPoseDecoderLe32
"TcpPoseDecoderLe32"
BEGIN
END_DATA_BLOCK

DATA_BLOCK "InstTcpTarget"   // DB13
{ S7_Optimized_Access := 'TRUE' }
VERSION : 0.1
// stored: InstanceOfName TcpTarget
"TcpTarget"
BEGIN
END_DATA_BLOCK

// folder: 40. Safety/F-Program

DATA_BLOCK "Main_Safety_RTG1_DB"   // DB1, F_DB
{ S7_Optimized_Access := 'TRUE' }
NAME : FUSI
VERSION : 0.1
// stored: InstanceOfName Main_Safety_RTG1
"Main_Safety_RTG1"
BEGIN
END_DATA_BLOCK

// folder: Eliminar

DATA_BLOCK "DB_Supervisor"   // DB9
{ S7_Optimized_Access := 'TRUE' }
VERSION : 0.1
   VAR
      Common : Struct
         plc_ok : Bool;
         supervisor_ok : Bool;
         system_ok : Bool;
         safety_ok : Bool;
         air_ok : Bool;
         insp_water_ok : Bool;
         tank_water_ok : Bool;
         robot_ok : Bool;
         step_plc : Int;
         step_supervisor : Int;
         error : Bool;
         reset_req : Bool;
      END_STRUCT;
      Identification : Struct   // pag 2
         carriage_id_req : Bool;   // Sup->PLC
         new_carriage_id : Bool;   // PLC->Sup
         id_req : Bool;   // Sup->PLC
         id_running : Bool;   // PLC->Sup
         id_ok : Bool;   // PLC->Sup
         teach_req : Bool;   // Sup->PLC
         system_ok : Bool;   // PLC->Sup (parte de id_ok)
         pa_check_req : Bool;   // Sup->PLC
         tcg_req : Bool;   // Sup->PLC
      END_STRUCT;
      Teaching : Struct   // pag 3
         teach_ready : Bool;   // PLC->Sup
         teach_running : Bool;   // Sup->PLC
         teach_state : Bool;   // Sup->PLC
         jump_start_us : Bool;   // PLC->Sup
      END_STRUCT;
      StartUs : Struct   // pag 4
         start_us_ready : Bool;   // PLC->Sup
         start_us_running : Bool;   // Sup->PLC
         start_us_state : Bool;   // Sup->PLC
      END_STRUCT;
      PACheck : Struct   // pag 5
         pa_check_ready : Bool;   // PLC->Sup
         elem_running : Bool;   // Sup->PLC
         elem_state : Bool;   // Sup->PLC
         bal_running : Bool;   // Sup->PLC
         bal_state : Bool;   // Sup->PLC
      END_STRUCT;
      Gain : Struct
         gain_ready : Bool;
         gain_running : Bool;
         gain_state : Bool;
      END_STRUCT;
      TCG_Check : Struct
         tcg_ready : Bool;
         tcg_running : Bool;
         tcg_next_step : Bool;
         jump_acq_ref : Bool;
         jump_tcg_adj : Bool;
      END_STRUCT;
      TCG_Adjust : Struct
         tcg_ready : Bool;
         jump_ref_acq : Bool;
      END_STRUCT;
      RefScan_Acq : Struct
         scan_ref_ready : Bool;
         scan_ref_running : Bool;
      END_STRUCT;
      InspScan : Struct
         scan_insp_ready : Bool;
         scan_insp_running : Bool;
         scan_insp_state : Bool;
         jump_ref_insp : Bool;
      END_STRUCT;
      RefScan_Verif : Struct
         scan_ref_ready : Bool;
         scan_ref_running : Bool;
         jump_start : Bool;
      END_STRUCT;
      Marking : Struct
         mark_req : Bool;
         mark_running : Bool;
         mark_state : Bool;
         jump_start : Bool;
         point_coordinates : Struct
            x : Real;
            y : Real;
            z : Real;
            "a" : Real;
            "b" : Real;
            c : Real;
         END_STRUCT;
      END_STRUCT;
   END_VAR
BEGIN
END_DATA_BLOCK

// folder: 10. System

FUNCTION_BLOCK "SeqManager"   // FB20, LAD
{ S7_Optimized_Access := 'TRUE' }
VERSION : 0.1
   VAR_INPUT
      systemArmed : Bool;
      autoBusy : Bool;
      servBusy : Bool;
      teachingRunning : Bool;
      startUsRunning : Bool;
      modeRequest : UInt;
      modeReqSeq : UInt;
   END_VAR
   VAR_OUTPUT
      modeEffective : UInt;
      modeReady : Bool;
      enterService : Bool;
      enterAuto : Bool;
   END_VAR
   VAR
      lastSeq : UInt;
      safeAllOk : Bool;
      windowAuto : Bool;
      acceptSrv : Bool;
      acceptAuto : Bool;
   END_VAR
BEGIN

REGION Network 1 (SCL)
   #safeAllOk := #systemArmed;
   // Ventana AUTO: OR de todos los *_running (ver tablas por etapa en el PDF).  // nivel sostenido
   #windowAuto :=
   #teachingRunning OR #startUsRunning;

   #enterService := FALSE;
   #enterAuto := FALSE;
   #acceptSrv := FALSE;
   #acceptAuto := FALSE;
END_REGION

REGION Network 2 (SCL)
   // 1) Nueva petición por contador
   IF #modeReqSeq <> #lastSeq THEN
       #lastSeq := #modeReqSeq;

       CASE #modeRequest OF
           0:  // SERVICE
               IF #safeAllOk AND (NOT #autoBusy) AND (NOT #windowAuto) THEN
                   #acceptSrv := TRUE;
               END_IF;

           1:  // AUTO
               IF #safeAllOk AND (NOT #servBusy) THEN
                   #acceptAuto := TRUE;
               END_IF;

       END_CASE;
   END_IF;
END_REGION

REGION Network 3 (SCL)
   IF #acceptSrv THEN
       #modeEffective := 0;
       #enterService := TRUE;
   ELSIF #acceptAuto THEN
       #modeEffective := 1;
       #enterAuto := TRUE;
   END_IF;

   // 3) Ready hacia HMI
   IF #modeEffective = 0 THEN
       #modeReady := #safeAllOk AND (NOT #autoBusy);
   ELSE
       #modeReady := #safeAllOk AND (NOT #servBusy);
   END_IF;
END_REGION
END_FUNCTION_BLOCK

FUNCTION_BLOCK "KukaControlSeq"   // FB21, LAD
{ S7_Optimized_Access := 'TRUE' }
VERSION : 0.1
BEGIN

REGION Network 1: Envia posiciones a la aplicacion KukaControl
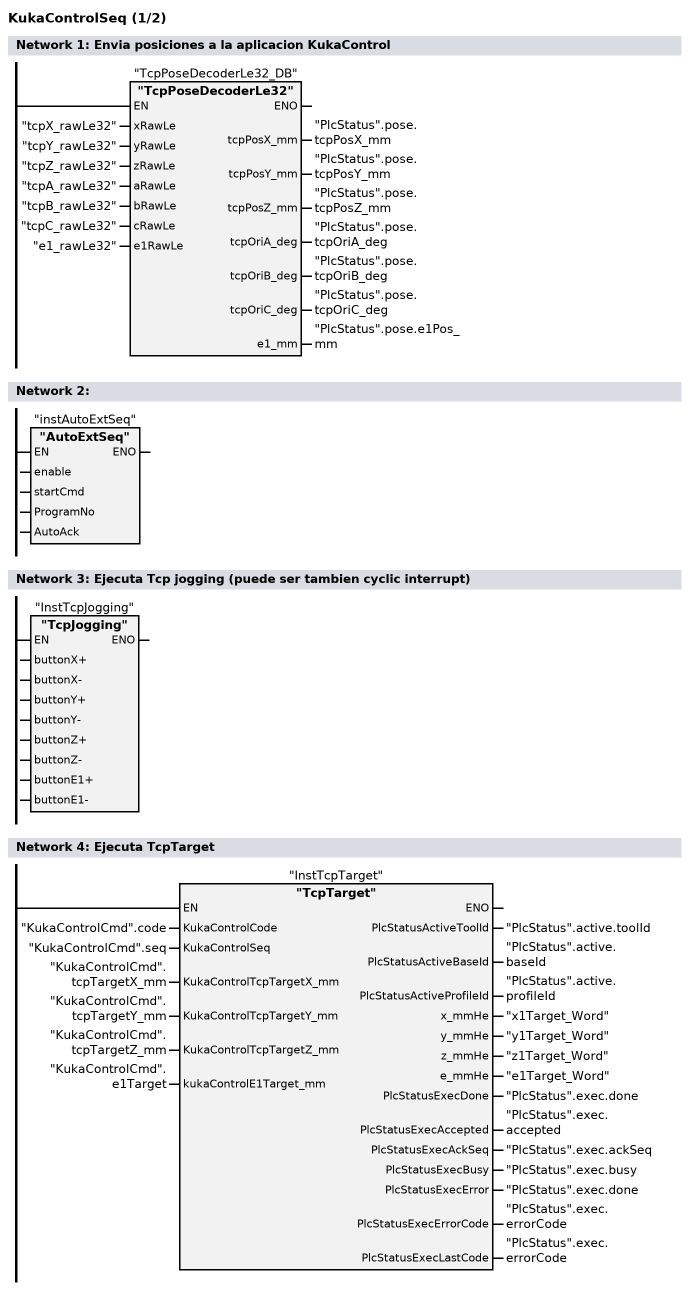
   RUNG wire#powerrail
      "TcpPoseDecoderLe32_DB"(xRawLe := "tcpX_rawLe32", yRawLe := "tcpY_rawLe32", zRawLe := "tcpZ_rawLe32", aRawLe := "tcpA_rawLe32", bRawLe := "tcpB_rawLe32", cRawLe := "tcpC_rawLe32", e1RawLe := "e1_rawLe32", tcpPosX_mm => "PlcStatus".pose.tcpPosX_mm, tcpPosY_mm => "PlcStatus".pose.tcpPosY_mm, tcpPosZ_mm => "PlcStatus".pose.tcpPosZ_mm, tcpOriA_deg => "PlcStatus".pose.tcpOriA_deg, tcpOriB_deg => "PlcStatus".pose.tcpOriB_deg, tcpOriC_deg => "PlcStatus".pose.tcpOriC_deg, e1_mm => "PlcStatus".pose.e1Pos_mm)
   END_RUNG
   // the same network as SCL:
   "TcpPoseDecoderLe32_DB"(xRawLe := "tcpX_rawLe32",   // "TcpPoseDecoderLe32"
                           yRawLe := "tcpY_rawLe32",
                           zRawLe := "tcpZ_rawLe32",
                           aRawLe := "tcpA_rawLe32",
                           bRawLe := "tcpB_rawLe32",
                           cRawLe := "tcpC_rawLe32",
                           e1RawLe := "e1_rawLe32",
                           tcpPosX_mm => "PlcStatus".pose.tcpPosX_mm,
                           tcpPosY_mm => "PlcStatus".pose.tcpPosY_mm,
                           tcpPosZ_mm => "PlcStatus".pose.tcpPosZ_mm,
                           tcpOriA_deg => "PlcStatus".pose.tcpOriA_deg,
                           tcpOriB_deg => "PlcStatus".pose.tcpOriB_deg,
                           tcpOriC_deg => "PlcStatus".pose.tcpOriC_deg,
                           e1_mm => "PlcStatus".pose.e1Pos_mm);
END_REGION

REGION Network 2
   RUNG wire#powerrail
      "instAutoExtSeq"(enable :=, startCmd :=, ProgramNo :=, AutoAck :=)
   END_RUNG
   // the same network as SCL:
   "instAutoExtSeq"();   // "AutoExtSeq"
END_REGION

REGION Network 3: Ejecuta Tcp jogging (puede ser tambien cyclic interrupt)
   RUNG wire#powerrail
      "InstTcpJogging"("buttonX+" :=, "buttonX-" :=, "buttonY+" :=, "buttonY-" :=, "buttonZ+" :=, "buttonZ-" :=, "buttonE1+" :=, "buttonE1-" :=)
   END_RUNG
   // the same network as SCL:
   "InstTcpJogging"();   // "TcpJogging"
END_REGION

REGION Network 4: Ejecuta TcpTarget
   RUNG wire#powerrail
      "InstTcpTarget"(KukaControlCode := "KukaControlCmd".code, KukaControlSeq := "KukaControlCmd".seq, KukaControlTcpTargetX_mm := "KukaControlCmd".tcpTargetX_mm, KukaControlTcpTargetY_mm := "KukaControlCmd".tcpTargetY_mm, KukaControlTcpTargetZ_mm := "KukaControlCmd".tcpTargetZ_mm, kukaControlE1Target_mm := "KukaControlCmd".e1Target, PlcStatusActiveToolId => "PlcStatus".active.toolId, PlcStatusActiveBaseId => "PlcStatus".active.baseId, PlcStatusActiveProfileId => "PlcStatus".active.profileId, x_mmHe => "x1Target_Word", y_mmHe => "y1Target_Word", z_mmHe => "z1Target_Word", e_mmHe => "e1Target_Word", PlcStatusExecDone => "PlcStatus".exec.done, PlcStatusExecAccepted => "PlcStatus".exec.accepted, PlcStatusExecAckSeq => "PlcStatus".exec.ackSeq, PlcStatusExecBusy => "PlcStatus".exec.busy, PlcStatusExecError => "PlcStatus".exec.done, PlcStatusExecErrorCode => "PlcStatus".exec.errorCode, PlcStatusExecLastCode => "PlcStatus".exec.errorCode)
   END_RUNG
   // the same network as SCL:
   "InstTcpTarget"(KukaControlCode := "KukaControlCmd".code,   // "TcpTarget"
                   KukaControlSeq := "KukaControlCmd".seq,
                   KukaControlTcpTargetX_mm := "KukaControlCmd".tcpTargetX_mm,
                   KukaControlTcpTargetY_mm := "KukaControlCmd".tcpTargetY_mm,
                   KukaControlTcpTargetZ_mm := "KukaControlCmd".tcpTargetZ_mm,
                   kukaControlE1Target_mm := "KukaControlCmd".e1Target,
                   PlcStatusActiveToolId => "PlcStatus".active.toolId,
                   PlcStatusActiveBaseId => "PlcStatus".active.baseId,
                   PlcStatusActiveProfileId => "PlcStatus".active.profileId,
                   x_mmHe => "x1Target_Word",
                   y_mmHe => "y1Target_Word",
                   z_mmHe => "z1Target_Word",
                   e_mmHe => "e1Target_Word",
                   PlcStatusExecDone => "PlcStatus".exec.done,
                   PlcStatusExecAccepted => "PlcStatus".exec.accepted,
                   PlcStatusExecAckSeq => "PlcStatus".exec.ackSeq,
                   PlcStatusExecBusy => "PlcStatus".exec.busy,
                   PlcStatusExecError => "PlcStatus".exec.done,
                   PlcStatusExecErrorCode => "PlcStatus".exec.errorCode,
                   PlcStatusExecLastCode => "PlcStatus".exec.errorCode);
END_REGION

REGION Network 5
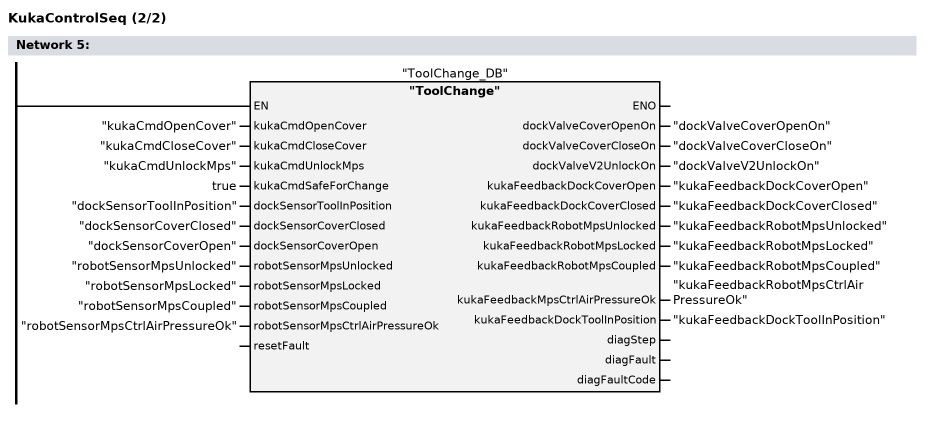
   RUNG wire#powerrail
      "ToolChange_DB"(kukaCmdOpenCover := "kukaCmdOpenCover", kukaCmdCloseCover := "kukaCmdCloseCover", kukaCmdUnlockMps := "kukaCmdUnlockMps", kukaCmdSafeForChange := true, dockSensorToolInPosition := "dockSensorToolInPosition", dockSensorCoverClosed := "dockSensorCoverClosed", dockSensorCoverOpen := "dockSensorCoverOpen", robotSensorMpsUnlocked := "robotSensorMpsUnlocked", robotSensorMpsLocked := "robotSensorMpsLocked", robotSensorMpsCoupled := "robotSensorMpsCoupled", robotSensorMpsCtrlAirPressureOk := "robotSensorMpsCtrlAirPressureOk", resetFault :=, dockValveCoverOpenOn => "dockValveCoverOpenOn", dockValveCoverCloseOn => "dockValveCoverCloseOn", dockValveV2UnlockOn => "dockValveV2UnlockOn", kukaFeedbackDockCoverOpen => "kukaFeedbackDockCoverOpen", kukaFeedbackDockCoverClosed => "kukaFeedbackDockCoverClosed", kukaFeedbackRobotMpsUnlocked => "kukaFeedbackRobotMpsUnlocked", kukaFeedbackRobotMpsLocked => "kukaFeedbackRobotMpsLocked", kukaFeedbackRobotMpsCoupled => "kukaFeedbackRobotMpsCoupled", kukaFeedbackMpsCtrlAirPressureOk => "kukaFeedbackRobotMpsCtrlAirPressureOk", kukaFeedbackDockToolInPosition => "kukaFeedbackDockToolInPosition", diagStep =>, diagFault =>, diagFaultCode =>)
   END_RUNG
   // the same network as SCL:
   "ToolChange_DB"(kukaCmdOpenCover := "kukaCmdOpenCover",   // "ToolChange"
                   kukaCmdCloseCover := "kukaCmdCloseCover",
                   kukaCmdUnlockMps := "kukaCmdUnlockMps",
                   kukaCmdSafeForChange := true,
                   dockSensorToolInPosition := "dockSensorToolInPosition",
                   dockSensorCoverClosed := "dockSensorCoverClosed",
                   dockSensorCoverOpen := "dockSensorCoverOpen",
                   robotSensorMpsUnlocked := "robotSensorMpsUnlocked",
                   robotSensorMpsLocked := "robotSensorMpsLocked",
                   robotSensorMpsCoupled := "robotSensorMpsCoupled",
                   robotSensorMpsCtrlAirPressureOk := "robotSensorMpsCtrlAirPressureOk",
                   dockValveCoverOpenOn => "dockValveCoverOpenOn",
                   dockValveCoverCloseOn => "dockValveCoverCloseOn",
                   dockValveV2UnlockOn => "dockValveV2UnlockOn",
                   kukaFeedbackDockCoverOpen => "kukaFeedbackDockCoverOpen",
                   kukaFeedbackDockCoverClosed => "kukaFeedbackDockCoverClosed",
                   kukaFeedbackRobotMpsUnlocked => "kukaFeedbackRobotMpsUnlocked",
                   kukaFeedbackRobotMpsLocked => "kukaFeedbackRobotMpsLocked",
                   kukaFeedbackRobotMpsCoupled => "kukaFeedbackRobotMpsCoupled",
                   kukaFeedbackMpsCtrlAirPressureOk => "kukaFeedbackRobotMpsCtrlAirPressureOk",
                   kukaFeedbackDockToolInPosition => "kukaFeedbackDockToolInPosition");
END_REGION
END_FUNCTION_BLOCK

FUNCTION_BLOCK "SupervisorSeq"   // FB22, LAD
{ S7_Optimized_Access := 'TRUE' }
VERSION : 0.1
   VAR
      firstScan : Bool;
      enteredStep : Bool;
      prev_step_plc : Int;
      prev_step_supervisor : Int;
      phase : Int;
      tcg_pos_index : Int;
      tcg_gate : Bool;
      cStep_IDENT : Int;
      cSTEP_TEACH : Int;
      cSTEP_STARTUS : Int;
      cSTEP_PA_CHECK : Int;
      cSTEP_GAIN : Int;
      cSTEP_TCG_CHECK : Int;
      cSTEP_TCG_ADJ : Int;
      cSTEP_REF_ACQ : Int;
      cSTEP_INSP : Int;
      cSTEP_REF_VERIF : Int;
      cSTEP_MARKING : Int;
   END_VAR
BEGIN

REGION Network 1 (SCL)
   IF #firstScan THEN
       "PlcStatus".Supervisor.global.plcOk := TRUE;


       "DB_Supervisor".Common.plc_ok := TRUE;
       "DB_Supervisor".Common.step_plc := #cStep_IDENT;
       #firstScan := FALSE;
   END_IF;

   "DB_Supervisor".Common.plc_ok := TRUE;


   // ---- State machine ----

   CASE "SupervisorCmd".global.stepSupervisor OF
           // 1) Identification (p.2)
       1:

           "DB_Supervisor".Identification.new_carriage_id :=
           "DB_Supervisor".Identification.carriage_id_req;

           CASE #phase OF
               0:
                   IF "DB_Supervisor".Identification.id_req THEN
                       "DB_Supervisor".Identification.id_running := TRUE;
                       "DB_Supervisor".Identification.id_ok :=
                       "DB_Supervisor".Common.safety_ok
                       AND "DB_Supervisor".Common.air_ok
                       AND "DB_Supervisor".Common.insp_water_ok
                       AND "DB_Supervisor".Common.tank_water_ok
                       AND "DB_Supervisor".Common.robot_ok
                       AND "DB_Supervisor".Common.supervisor_ok
                       AND "DB_Supervisor".Identification.system_ok;
                       #phase := 1;
                   END_IF;
               1:
                   "DB_Supervisor".Identification.id_running := FALSE;
                   IF "DB_Supervisor".Identification.id_ok THEN
                       IF "DB_Supervisor".Identification.teach_req THEN
                           "DB_Supervisor".Common.step_plc := 2;
                       ELSE
                           "DB_Supervisor".Common.step_plc := 3;
                       END_IF;
                   END_IF;
           END_CASE;

           ;

           // 2) Teaching (p.3)
       2:

           CASE  #phase OF
               0:
                   "DB_Supervisor".Teaching.teach_ready := TRUE;
                   IF "DB_Supervisor".Teaching.teach_running THEN
                       "DB_Supervisor".Teaching.teach_ready := FALSE;
                       #phase := 1;
                   END_IF;
               1:
                   IF NOT "DB_Supervisor".Teaching.teach_running THEN
                       IF "DB_Supervisor".Teaching.teach_state THEN
                           "DB_Supervisor".Common.step_plc := 3;
                       END_IF;
                   END_IF;
           END_CASE;


           // 3) Start US (p.4)
           3:

           CASE #phase OF
               0:
                   "DB_Supervisor".StartUs.start_us_ready := TRUE;
                   IF "DB_Supervisor".StartUs.start_us_running THEN
                       "DB_Supervisor".StartUs.start_us_ready := FALSE;
                       #phase := 1;
                   END_IF;
               1:
                   IF NOT "DB_Supervisor".StartUs.start_us_running THEN
                       IF "DB_Supervisor".StartUs.start_us_state THEN
                           IF "DB_Supervisor".Identification.pa_check_req THEN
                               "DB_Supervisor".Common.step_plc := 4;
                           ELSE
                               "DB_Supervisor".Common.step_plc := 5;
                           END_IF;
                       END_IF;
                   END_IF;
           END_CASE;


           // 4) PA‑Check (p.5)
           4:

           CASE #phase OF
               0:
                   "DB_Supervisor".PACheck.pa_check_ready := TRUE;
                   IF "DB_Supervisor".PACheck.elem_running THEN
                       "DB_Supervisor".PACheck.pa_check_ready := FALSE;
                       #phase := 1;
                   END_IF;
               1:
                   IF NOT "DB_Supervisor".PACheck.elem_running THEN
                       IF "DB_Supervisor".PACheck.elem_state THEN
                           #phase := 2;
                       END_IF;
                   END_IF;
               2:
                   IF "DB_Supervisor".PACheck.bal_running THEN
                       #phase := 3;
                   END_IF;
               3:
                   IF NOT "DB_Supervisor".PACheck.bal_running THEN
                       IF "DB_Supervisor".PACheck.bal_state THEN
                           "DB_Supervisor".Common.step_plc := 5;
                       END_IF;
                   END_IF;
           END_CASE;


           // 5) Gain (p.6)
           5:

           CASE #phase OF
               0:
                   "DB_Supervisor".Gain.gain_ready := TRUE;
                   IF "DB_Supervisor".Gain.gain_running THEN
                       "DB_Supervisor".Gain.gain_ready := FALSE;
                       #phase := 1;
                   END_IF;
               1:
                   IF NOT "DB_Supervisor".Gain.gain_running THEN
                       IF "DB_Supervisor".Gain.gain_state THEN
                           IF "DB_Supervisor".Identification.tcg_req THEN
                               "DB_Supervisor".Common.step_plc := 6;
                           ELSE
                               "DB_Supervisor".Common.step_plc := 8;
                           END_IF;
                       END_IF;
                   END_IF;
           END_CASE;


           // 6) TCG Check (p.7)
           6:

           CASE #phase OF
               0:
                   "DB_Supervisor".TCG_Check.tcg_ready := TRUE;
                   #tcg_pos_index := 0;
                   IF "DB_Supervisor".TCG_Check.tcg_running THEN
                       "DB_Supervisor".TCG_Check.tcg_ready := FALSE;
                       #phase := 1;
                   END_IF;

               1: // gate a tcg_next_step
                   IF "DB_Supervisor".TCG_Check.tcg_next_step AND NOT #tcg_gate THEN
                       #tcg_gate := TRUE;
                       #tcg_pos_index := #tcg_pos_index + 1; // 1..3
                   END_IF;
                   IF NOT "DB_Supervisor".TCG_Check.tcg_next_step THEN
                       #tcg_gate := FALSE;
                   END_IF;

                   IF NOT "DB_Supervisor".TCG_Check.tcg_running THEN
                       #phase := 2;
                   END_IF;

               2:
                   IF #tcg_pos_index >= 3 THEN
                       IF "DB_Supervisor".TCG_Check.jump_acq_ref THEN
                           "DB_Supervisor".Common.step_plc := 8;
                       ELSIF "DB_Supervisor".TCG_Check.jump_tcg_adj THEN
                           "DB_Supervisor".Common.step_plc := 7;
                       END_IF;
                   END_IF;
           END_CASE;


           // 7) TCG Adjust (p.7)
           7:

           CASE #phase OF
               0:
                   "DB_Supervisor".TCG_Adjust.tcg_ready := TRUE;
                   #phase := 1;
               1:
                   IF "DB_Supervisor".TCG_Adjust.jump_ref_acq THEN
                       "DB_Supervisor".Common.step_plc := 8;
                   END_IF;
           END_CASE;


           // 8) RefScan – Acquisition (p.8)
           8:

           CASE #phase OF
               0:
                   "DB_Supervisor".RefScan_Acq.scan_ref_ready := TRUE;
                   IF "DB_Supervisor".RefScan_Acq.scan_ref_running THEN
                       "DB_Supervisor".RefScan_Acq.scan_ref_ready := FALSE;
                       #phase := 1;
                   END_IF;
               1:
                   IF NOT "DB_Supervisor".RefScan_Acq.scan_ref_running THEN
                       "DB_Supervisor".Common.step_plc := 9;
                   END_IF;
           END_CASE;


           // 9) Inspection Scan (p.9)
           9:

           CASE #phase OF
               0:
                   "DB_Supervisor".InspScan.scan_insp_ready := TRUE;
                   IF "DB_Supervisor".InspScan.scan_insp_running THEN
                       "DB_Supervisor".InspScan.scan_insp_ready := FALSE;
                       #phase := 1;
                   END_IF;
               1:
                   IF "DB_Supervisor".InspScan.jump_ref_insp THEN
                       "DB_Supervisor".Common.step_plc := 10;
                   END_IF;
           END_CASE;


           // 10) RefScan – Verification (p.10)
           10:

           CASE #phase OF
               0:
                   "DB_Supervisor".RefScan_Verif.scan_ref_ready := TRUE;
                   IF "DB_Supervisor".RefScan_Verif.scan_ref_running THEN
                       "DB_Supervisor".RefScan_Verif.scan_ref_ready := FALSE;
                       #phase := 1;
                   END_IF;
               1:
                   IF "DB_Supervisor".RefScan_Verif.jump_start THEN
                       "DB_Supervisor".Common.step_plc := 1;
                   END_IF;
           END_CASE;

           // 11) Marking / Pre‑evaluation (p.11)
           11:

           CASE #phase OF
               0:
                   IF "DB_Supervisor".Marking.mark_req THEN
                       "DB_Supervisor".Marking.mark_running := TRUE;
                       #phase := 1;
                   END_IF;
               1:
                   // Sustituir por DONE real:
                   IF TRUE THEN
                       "DB_Supervisor".Marking.mark_running := FALSE;
                       "DB_Supervisor".Marking.mark_state := TRUE;
                       #phase := 2;
                   END_IF;
               2:
                   IF "DB_Supervisor".Marking.jump_start THEN
                       "DB_Supervisor".Common.step_plc := 1;
                   END_IF;
           END_CASE;


       ELSE
           "DB_Supervisor".Common.step_plc := 1;
       END_CASE;
END_REGION
END_FUNCTION_BLOCK

ORGANIZATION_BLOCK "Main"   // OB1, LAD, ProgramCycle
TITLE = "Main Program Sweep (Cycle)"
{ S7_Optimized_Access := 'TRUE' }
VERSION : 0.1
   VAR_INPUT
      Initial_Call : Bool;   // Initial call of this OB
      Remanence : Bool;   // =True, if remanent data are available
   END_VAR
   VAR_TEMP
      evtEnterSrv : Bool;   // // Eventos de modo service jog
      evtEnterAuto : Bool;   // // Eventos de modo auto
      muxSelStb : Bool;
      muxStartStb : Bool;
      muxPgno : Byte;
      u : UDInt;
   END_VAR
BEGIN

REGION Network 1 (SCL): // ====================== READ (%I) ======================
   // // —— Enlaza estos símbolos a tus %I en el árbol de dispositivos ——
   //   // EStop_DI, SafeDoor_DI, AirPressure_DI, WaterInsp_DI, WaterTank_DI, RobotReady_DI, ...
END_REGION

REGION Network 2: // 1) Árbitro de modo: decide y emite
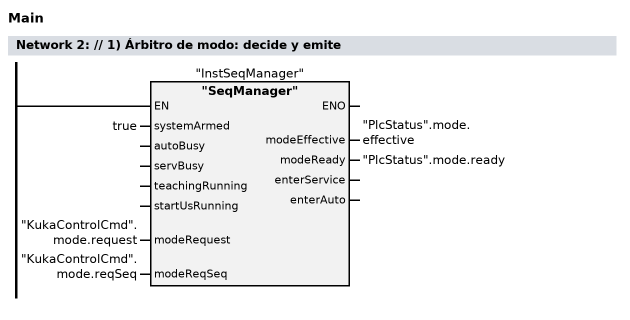
   RUNG wire#powerrail
      "InstSeqManager"(systemArmed := true, autoBusy :=, servBusy :=, teachingRunning :=, startUsRunning :=, modeRequest := "KukaControlCmd".mode.request, modeReqSeq := "KukaControlCmd".mode.reqSeq, modeEffective => "PlcStatus".mode.effective, modeReady => "PlcStatus".mode.ready, enterService =>, enterAuto =>)
   END_RUNG
   // the same network as SCL:
   "InstSeqManager"(systemArmed := true,   // "SeqManager"
                    modeRequest := "KukaControlCmd".mode.request,
                    modeReqSeq := "KukaControlCmd".mode.reqSeq,
                    modeEffective => "PlcStatus".mode.effective,
                    modeReady => "PlcStatus".mode.ready);
END_REGION

REGION Network 3 (SCL): // 2) Ejecuta o service o Auto
       IF "PlcStatus".mode.effective = 1 THEN
           // SUPERVISOR : Mode Effective = 1
           "InstSupervisorSeq"();
       ELSE
           // KUKACONTROL: Mode Effective = 0
           "InstKukaControlSeq"();
       END_IF;
END_REGION
END_ORGANIZATION_BLOCK

// folder: 10. System/Utilities

FUNCTION_BLOCK "ClockPulse"   // FB67, LAD
{ S7_Optimized_Access := 'TRUE' }
VERSION : 0.1
BEGIN
END_FUNCTION_BLOCK

// folder: 20. Robot Services/AutoExt

FUNCTION_BLOCK "AutoExtSeq"   // FB31, LAD
{ S7_Optimized_Access := 'TRUE' }
VERSION : 0.1
   VAR_INPUT
      enable : Bool;   // // habilita interfaz
      startCmd : Bool;   // // flanco de arranque
      ProgramNo : Byte;   // / nº CASE (1..255)
      AutoAck : Bool;   // // auto-confirmar STOPMESS
   END_VAR
   VAR
      rStart : R_TRIG;
      Static_1 : Bool;
      fReq : F_TRIG;
      pending : Bool;   // // hay pedido en curso
      running : Bool;   // // PRO_ACT latcheado
      pgnoLat : Byte;   // // PGNO latcheado
      tpStart : TP_TIME;
      tpAck : TP_TIME;
      rStop : R_TRIG;
   END_VAR
BEGIN

REGION Network 1 (SCL)
   // ---- habilitaciones fijas ----
   //%QX601.7 := Enable;        // I_O_ACT
   //%QX601.3 := Enable;              // MOVE_ENABLE
   //%QX601.5 := Enable;        // DRIVES_ON
   //%QX601.6 := NOT %QX601.5;       // DRIVES_OFF (invertido)
END_REGION

REGION Network 2 (SCL): // ---- detectar solicitud de arranque ----
   #rStart(CLK:=#startCmd);
   IF #rStart.Q AND NOT #pending AND NOT "tcpPosX_02" THEN
       #pending := TRUE;
       #pgnoLat := #ProgramNo;
     //  "Tag_5" := #pgnoLat;         // escribir PGNO (8 bits)
   END_IF;
END_REGION

REGION Network 3 (SCL): Paridad
   // ---- paridad (EVEN) ----
   //"tcpTargetX_08" := FC_EvenParity(b := #pgnoLat);
END_REGION

REGION Network 4 (SCL): // ---- VALID solo mientras PGNO_REQ=1 y hay pedido ----
   IF #pending THEN
       "tcpTargetX_09" := "tcpPosX_01";       // seguir a PGNO_REQ
       //  %QX601.1 := %IX600.1;       // seguir a PGNO_REQ
   ELSE
       "tcpTargetX_09" := FALSE;
       //  %QX601.1 := FALSE;
   END_IF;
END_REGION

REGION Network 5 (SCL): // ---- cuando PGNO_REQ baja -> pulso de EXT_START ---
   #fReq(CLK := "tcpPosX_05");
   #tpStart(IN := (#pending AND #fReq.Q),
            PT := T#120ms);
   "tcpTargetX_10" := #tpStart.Q;
END_REGION

REGION Network 6 (SCL): // ---- auto-confirmar mensajes cuando aparezcan ----
   #rStop(CLK := "tcpPosX_05");
   #tpAck(IN := (#AutoAck AND #rStop.Q),
          PT := T#120ms);
   "tcpTargetX_12" := #tpAck.Q;
END_REGION

REGION Network 7 (SCL): ---- seguimiento de ejecución y liberación de 'pending' ----
   IF "tcpPosX_02" THEN             // PRO_ACT=1
       #running := TRUE;
   ELSIF #running AND NOT "tcpPosX_02" THEN
       #running := FALSE;
       #pending := FALSE;        // ciclo terminado
   END_IF;
END_REGION
END_FUNCTION_BLOCK

// folder: 20. Robot Services/Mov Manual

FUNCTION_BLOCK "TcpJogging"   // FB5, LAD
{ S7_Optimized_Access := 'TRUE' }
VERSION : 0.1
   VAR_INPUT
      "buttonX+" : Bool;
      "buttonX-" : Bool;
      "buttonY+" : Bool;
      "buttonY-" : Bool;
      "buttonZ+" : Bool;
      "buttonZ-" : Bool;
      "buttonE1+" : Bool;
      "buttonE1-" : Bool;
   END_VAR
BEGIN

REGION Network 1 (SCL): Mapea los valores de los botones de WF
   IF "PlcStatus".mode.effective = 0 THEN

       "Tag_1" := TRUE;
       //MOV X,Y,Z
       //%Q630.0 = buttonX+
       //%Q630.1 = buttonX-
       //%Q630.2 = buttonY+
       //%Q630.3 = buttonY-
       //%Q630.4 = buttonZ+
       //%Q630.5 = buttonZ-
       //MOV A,B,C
       //%Q630.6 = buttonWF +A
       //%Q630.7 = buttonWF -A
       //%Q631.0 = buttonWF +B
       //%Q631.1 = buttonWF -B
       //%Q631.2 = buttonWF +C
       //%Q631.3 = buttonWF -C
       //Mov E1
       //%Q631.4 = buttonWF +E1
       //%Q631.5 = buttonWF -E1

   ELSE
       //%Q631.1 = buttonWF -B
       "Tag_1" := FALSE;
   END_IF;
END_REGION
END_FUNCTION_BLOCK

FUNCTION_BLOCK "TcpTarget"   // FB11, LAD
{ S7_Optimized_Access := 'TRUE' }
VERSION : 0.1
   VAR_INPUT
      KukaControlCode : UInt;
      KukaControlSeq : UInt;
      KukaControlTcpTargetX_mm : LReal;
      KukaControlTcpTargetY_mm : LReal;
      KukaControlTcpTargetZ_mm : LReal;
      kukaControlE1Target_mm : LReal;
   END_VAR
   VAR_OUTPUT
      PlcStatusActiveToolId : UInt;
      PlcStatusActiveBaseId : UInt;
      PlcStatusActiveProfileId : UInt;
      x_mmHe : DWord;
      y_mmHe : DWord;
      z_mmHe : DWord;
      e_mmHe : DWord;
      PlcStatusExecDone : Bool;
      PlcStatusExecAccepted : Bool;
      PlcStatusExecAckSeq : UInt;
      PlcStatusExecBusy : Bool;
      PlcStatusExecError : Bool;
      PlcStatusExecErrorCode : DWord;
      PlcStatusExecLastCode : UInt;
   END_VAR
   VAR
      lastMoveSeq : Word;
      state : Int;
      tmoMove : TON_TIME;
      rbDoneEdge : R_TRIG;
   END_VAR
   VAR_TEMP
      x_dint : DInt;
      y_dint : DInt;
      z_dint : DInt;
      n_dint : DInt;
      code_int : UInt;
   END_VAR
BEGIN

REGION Network 1 (SCL)

   CASE #state OF
       0: // IDLE -> GO == ACK
           #"PlcStatusExecAccepted" := FALSE;
           #"PlcStatusExecBusy" := FALSE;
           #"PlcStatusExecError" := FALSE;
           #PlcStatusExecDone := FALSE;


           // Nuevo comando si llega seq distinto y hay código válido
           IF (#KukaControlSeq <> #lastMoveSeq)  THEN

               IF ("goTrigger" = "rbDone") THEN
                   // 1) Volcar dataset PNIO (tool/base/vel/target...) hacia el robot
                   // Prepara dataset hacia KUKA

                   //  Primero: Escalar mm → entero (µm). Ajusta el redondeo si lo prefieres TRUNC, FLOOR, etc.
                   #code_int := #KukaControlCode;
                   // 1) Usa el code local (sin swap) para decidir

                   IF #code_int = 130 THEN
                       //  Primero: Escalar mm → entero (µm). Ajusta el redondeo si lo prefieres TRUNC, FLOOR, etc.
                       #n_dint := LREAL_TO_DINT(ROUND(#"kukaControlE1Target_mm"));
                       // Segundo Convertir a DWORD y hacer SWAP para que el KRC lo lea correctamente
                       #e_mmHe := SWAP(DINT_TO_DWORD(#n_dint));
                   END_IF;

                   IF #code_int = 101 THEN
                       //  Primero: Escalar mm → entero (µm). Ajusta el redondeo si lo prefieres TRUNC, FLOOR, etc.
                       #x_dint := LREAL_TO_DINT(ROUND(#"KukaControlTcpTargetX_mm"));
                       // Segundo Convertir a DWORD y hacer SWAP para que el KRC lo lea correctamente
                       #x_mmHe := SWAP(DINT_TO_DWORD(#x_dint));
                   END_IF;

                   IF #code_int = 102 THEN
                       //  Primero: Escalar mm → entero (µm). Ajusta el redondeo si lo prefieres TRUNC, FLOOR, etc.
                       #y_dint := LREAL_TO_DINT(ROUND(#"KukaControlTcpTargetY_mm"));
                       // Segundo Convertir a DWORD y hacer SWAP para que el KRC lo lea correctamente
                       #y_mmHe := SWAP(DINT_TO_DWORD(#y_dint));
                   END_IF;

                   IF #code_int = 103 THEN
                       //  Primero: Escalar mm → entero (µm). Ajusta el redondeo si lo prefieres TRUNC, FLOOR, etc.
                       #z_dint := LREAL_TO_DINT(ROUND(#"KukaControlTcpTargetZ_mm"));
                       // Segundo Convertir a DWORD y hacer SWAP para que el KRC lo lea correctamente
                       #z_mmHe := SWAP(DINT_TO_DWORD(#z_dint));
                   END_IF;

                   // Segundo Convertir a DWORD y hacer SWAP para que el KRC lo lea correctamente
                   "moveCodeKuka" := SWAP(UINT_TO_WORD(#code_int));

                   "goTrigger" := NOT "goTrigger";     // Dispara pedido
                   #lastMoveSeq := #KukaControlSeq;          // <-- memoriza!
                   #state := 20;                    // BUSY
                   // Aún ocupado (no debería ocurrir si sigues la regla)
               END_IF;

           END_IF;

       20: // BUSY

           #"PlcStatusExecBusy" := TRUE;
           IF ("rbDone" = "goTrigger") THEN
               // Robot ya igualó ACK a GO -> terminó
               "PlcStatus".exec.done := TRUE;
               #state := 0;                         // vuelve a IDLE
           END_IF;

       30: // DONE
           // limpiar y volver a IDLE
           #state := 0;


   END_CASE;
END_REGION
END_FUNCTION_BLOCK

// folder: 20. Robot Services/RobotPos

FUNCTION_BLOCK "TcpPoseDecoderLe32"   // FB4, LAD
{ S7_Optimized_Access := 'TRUE' }
VERSION : 0.1
// Decodifica con SWAP, convierte a DINT y escala.
   VAR_INPUT
      xRawLe : DWord;
      yRawLe : DWord;
      zRawLe : DWord;
      aRawLe : DWord;
      bRawLe : DWord;
      cRawLe : DWord;
      e1RawLe : DWord;
   END_VAR
   VAR_OUTPUT
      tcpPosX_mm : LReal;
      tcpPosY_mm : LReal;
      tcpPosZ_mm : LReal;
      tcpOriA_deg : LReal;
      tcpOriB_deg : LReal;
      tcpOriC_deg : LReal;
      e1_mm : LReal;
   END_VAR
   VAR_TEMP
      xDint : DInt;
      yDint : DInt;
      zDint : DInt;
      aDint : DInt;
      bDint : DInt;
      cDint : DInt;
      e1Dint : DInt;
   END_VAR
BEGIN

REGION Network 1 (SCL): // 1) Endianness: ABCD -> DCBA
   #xDint := DWORD_TO_DINT(SWAP(#xRawLe));
   #yDint := DWORD_TO_DINT(SWAP(#yRawLe));
   #zDint := DWORD_TO_DINT(SWAP(#zRawLe));
   #aDint := DWORD_TO_DINT(SWAP(#aRawLe));
   #bDint := DWORD_TO_DINT(SWAP(#bRawLe));
   #cDint := DWORD_TO_DINT(SWAP(#cRawLe));
   #e1Dint := DWORD_TO_DINT(SWAP(#e1RawLe));
END_REGION

REGION Network 2 (SCL): // 2) Escala fixed-point: µm->mm, mdeg->deg
   #tcpPosX_mm := DINT_TO_LREAL(#xDint) / 1000.0;
   #tcpPosY_mm := DINT_TO_LREAL(#yDint) / 1000.0;
   #tcpPosZ_mm := DINT_TO_LREAL(#zDint) / 1000.0;
   #tcpOriA_deg := DINT_TO_LREAL(#aDint) / 1000.0;
   #tcpOriB_deg := DINT_TO_LREAL(#bDint) / 1000.0;
   #tcpOriC_deg := DINT_TO_LREAL(#cDint) / 1000.0;
   #e1_mm := DINT_TO_LREAL(#e1Dint) / 1000.0;  // mm o deg según tu E1
END_REGION
END_FUNCTION_BLOCK

// folder: 20. Robot Services/Tooling & Parking

FUNCTION_BLOCK "ToolChange"   // FB6, LAD
TITLE = FB: ManageTed009Station
{ S7_Optimized_Access := 'TRUE' }
VERSION : 0.1
// //  - KUKA manda órdenes (kukaCmd*)
// //  - El FB acciona bobinas de la docking (dockValve*On)
// //  - El FB publica ecos/estados para el KUKA (kukaFeedback*)
// //  - V2 (Unlock) puede mantenerse automática con útil aparcado
// //    (AutoUnlockWhenToolPresent = TRUE) [REF: estándar automático]. 
// //    Con útil ausente, no se activa para evitar soplado innecesario.
// //  - Tapa: FSM con interlock de zona segura y timeouts simétricos.
// //  - Diagnóstico: diagStep/diagFault/diagFaultCode.
// //
// //  Referencias (ver manual Stäubli TED009):
// //    • Sequence plan y sondeo ~20 ms durante conectar/desconectar. 
// //    • +21 mm: E2=0 ∧ E3=1 ∧ D1=0 antes de acoplar. 
// //    • z=0: bloquear retirando V2 y esperar E2=1 ∧ D1=1 (+E1=1). 
// //    • Retiradas +10/+70 y +25/>29 (comentadas para el programa del robot).
   VAR_INPUT
      kukaCmdOpenCover : Bool;
      kukaCmdCloseCover : Bool;
      kukaCmdUnlockMps : Bool;
      kukaCmdSafeForChange : Bool;
      dockSensorToolInPosition : Bool;   // E6
      dockSensorCoverClosed : Bool;   // E4
      dockSensorCoverOpen : Bool;   // E5
      robotSensorMpsUnlocked : Bool;   // E3
      robotSensorMpsLocked : Bool;   // E2
      robotSensorMpsCoupled : Bool;   // E1
      robotSensorMpsCtrlAirPressureOk : Bool;   // D1
      resetFault : Bool;
   END_VAR
   VAR_OUTPUT
      dockValveCoverOpenOn : Bool;   // bobina abrir tapa
      dockValveCoverCloseOn : Bool;   // bobina cerrar tapa
      dockValveV2UnlockOn : Bool;   // V2: aire de desbloqueo hacia módulo del robot
      kukaFeedbackDockCoverOpen : Bool;
      kukaFeedbackDockCoverClosed : Bool;
      kukaFeedbackRobotMpsUnlocked : Bool;
      kukaFeedbackRobotMpsLocked : Bool;
      kukaFeedbackRobotMpsCoupled : Bool;
      kukaFeedbackMpsCtrlAirPressureOk : Bool;
      kukaFeedbackDockToolInPosition : Bool;
      diagStep : Int;
      diagFault : Bool;
      diagFaultCode : Int;
   END_VAR
   VAR
      "step" : Int;
      fault : Bool;
      faultCode : Int;
      AutoUnlockWhenToolPresent : Bool := true;   // // modo auto
      coverTimeout : Time := T#8S;   // // timeout de tapa (abrir/cerrar)
      unlockTimeout : Time := T#2S;   // // timeout de UNLOCK (E3=1 & D1=0)
      unlockReq : Bool;
      unlockReqEnabled : Bool;
      tempCoverOpen : TON_TIME;
      tempCoverClose : TON_TIME;
      tempUnlock : TON_TIME;
      autoUnlockEligible : Bool;
   END_VAR
   VAR CONSTANT
      StateIdle : Int := 0;
      StateOpening : Int := 10;
      StateOpen : Int := 11;
      StateClosing : Int := 20;
      StateClosed : Int := 21;
      FaultNone : Int;
      FaultOpenTimeout : Int := 101;
      FaultCloseTimeout : Int := 102;
      FaultUnlockTimeout : Int := 201;
      FaultInterlock : Int := 301;
   END_VAR
BEGIN

REGION Network 1 (SCL): Lógica de tapa + V2 (Unlock) de la docking
   // --- Feedbacks de estados al robot (eco directo de sensores físicos)
   #kukaFeedbackDockToolInPosition := #dockSensorToolInPosition; // E6 - herramienta en docking station
   #kukaFeedbackDockCoverOpen := #dockSensorCoverOpen;         // E4 - tapa abierta
   #kukaFeedbackDockCoverClosed := #dockSensorCoverClosed;     // E5 - tapa cerrada
   #kukaFeedbackRobotMpsUnlocked := #robotSensorMpsUnlocked;  // E3 - MPS desbloqueado (robot side)
   #kukaFeedbackRobotMpsLocked := #robotSensorMpsLocked;     // E2 - MPS bloqueado (robot side
   #kukaFeedbackRobotMpsCoupled := #robotSensorMpsCoupled;        // E1 - MPS acoplado  (robot side) 
   #kukaFeedbackMpsCtrlAirPressureOk := #robotSensorMpsCtrlAirPressureOk;  // D1 -presostato módulo aire control (robot)

   // ---- Reset de fallos/estado -------------------------------------------
   // Permite reconocer fallos desde HMI/Robot. Pone las salidas a 0 y la FSM (flow state machine)
   // Deja el FB en reposo (IDLE), corta bobinas y reinicia tempor TONs.
   IF #resetFault THEN
       #fault := FALSE;
       #faultCode := #FaultNone;
       #step := #StateIdle;

       #dockValveCoverOpenOn := FALSE;
       #dockValveCoverCloseOn := FALSE;
       #dockValveV2UnlockOn := FALSE;

       // Reset explícito de TON: IN=FALSE + PT definido
       #tempCoverOpen(IN := FALSE,
                      PT := #coverTimeout);
       #tempCoverClose(IN := FALSE,
                       PT := #coverTimeout);
       #tempUnlock(IN := FALSE,
                   PT := #unlockTimeout);
   END_IF;

   // ================= LÓGICA DE TAPA (máquina de estados) =================
   // Interlock básico: no se permite accionar tapa si el robot no confirma zona segura
   // (manual: abrir/cerrar solo fuera del barrido).
   CASE #step OF

       #StateIdle: // IDLE
           // Reposo ( tapa sin accionar); evaluar órdenes de KUKA.
           #dockValveCoverOpenOn := FALSE;
           #dockValveCoverCloseOn := FALSE;

           IF #kukaCmdSafeForChange THEN
               // Abrir si lo pide el robot y aún no está abierta
               IF (#kukaCmdOpenCover AND NOT #dockSensorCoverOpen) THEN
                   #step := #StateOpening;
               END_IF;
               // Cerrar si lo pide el robot y aún no está cerrada
               IF (#kukaCmdCloseCover AND NOT #dockSensorCoverClosed) THEN
                   #step := #StateClosing;
               END_IF;
           ELSIF (#kukaCmdOpenCover OR #kukaCmdCloseCover) THEN
               // Petición sin zona segura -> fallo de interlock
               #fault := TRUE;
               #faultCode := #FaultInterlock; // robot no garantiza zona segura
           END_IF;

       #StateOpening:  // Abrir tapa
           #dockValveCoverOpenOn := TRUE;
           #dockValveCoverCloseOn := FALSE;

           // Timeout de apertura: si no llega "tapa abierta" dentro de coverTimeout -> fallo.
           // coverTimeout debe ser > 3 s (tiempo típico de maniobra)
           #tempCoverOpen(IN := NOT #dockSensorCoverOpen,
                          PT := #coverTimeout);

           IF (#dockSensorCoverOpen AND NOT #dockSensorCoverClosed) THEN
               #tempCoverOpen(IN := FALSE,
                              PT := #coverTimeout);
               #step := #StateOpen;
           ELSIF #tempCoverOpen.Q THEN
               #fault := TRUE;
               #faultCode := #FaultOpenTimeout;
               #dockValveCoverOpenOn := FALSE;
               #step := #StateIdle;
           END_IF;


       #StateOpen: // Tapa abierta (estable)
           #dockValveCoverOpenOn := FALSE;
           #dockValveCoverCloseOn := FALSE;

           IF (#kukaCmdSafeForChange AND #kukaCmdCloseCover) THEN
               #step := #StateClosing;
           END_IF;


       #StateClosing: // Cerrar tapa
           #dockValveCoverOpenOn := FALSE;
           #dockValveCoverCloseOn := TRUE;

           // Timeout de cierre: si no llega "tapa cerrada" dentro de coverTimeout -> fallo.
           #tempCoverClose(IN := NOT #dockSensorCoverClosed,
                           PT := #coverTimeout);

           IF (#dockSensorCoverClosed AND NOT #dockSensorCoverOpen) THEN
               #tempCoverClose(IN := FALSE,
                               PT := #coverTimeout);
               #step := #StateClosed;
           ELSIF #tempCoverClose.Q THEN
               #fault := TRUE;
               #faultCode := #FaultCloseTimeout;
               #dockValveCoverCloseOn := FALSE;
               #step := #StateIdle;
           END_IF;

       #StateClosed: // Tapa cerrada (estable)
           #dockValveCoverOpenOn := FALSE;
           #dockValveCoverCloseOn := FALSE;

           IF (#kukaCmdSafeForChange AND #kukaCmdOpenCover) THEN
               #step := #StateOpening;
           END_IF;

       ELSE
           #step := #StateIdle;
   END_CASE;

   // Exclusión mutua de bobinas de tapa (seguridad por si alguna rama dejó ambas a 1)
   IF #dockValveCoverOpenOn THEN
       #dockValveCoverCloseOn := FALSE;
   END_IF;
   IF #dockValveCoverCloseOn THEN
       #dockValveCoverOpenOn := FALSE;
   END_IF;


   // -------- Arbitraje de V2 (UNLOCK) --------
   // Auto válido solo si:
   //   - #AutoUnlockWhenToolPresent = TRUE (política activada)
   //   - #dockSensorToolInPosition = TRUE (herramienta aparcada)
   //   - #robotSensorMpsCoupled = FALSE (E1=0, aún NO acoplado)
   #autoUnlockEligible :=
   #AutoUnlockWhenToolPresent
   AND #dockSensorToolInPosition
   AND NOT #robotSensorMpsCoupled;

   // Prioridad al robot (su orden OR con el auto elegible).
   #dockValveV2UnlockOn := #kukaCmdUnlockMps OR #autoUnlockEligible;

   // Supervisión del estado desbloqueado (E3=1 y D1=0 en tiempo):
   #tempUnlock(
               IN := (#dockValveV2UnlockOn
               AND NOT (#robotSensorMpsUnlocked
               AND NOT #robotSensorMpsCtrlAirPressureOk)),
               PT := #unlockTimeout
   );
   IF NOT #dockValveV2UnlockOn THEN
       // reset explícito del TON cuando ya no se pide V2
       #tempUnlock(IN := FALSE,
                   PT := #unlockTimeout);
   END_IF;

   // -------------------- DIAGNÓSTICO PUBLICADO ----------------------------
   #diagStep := #step; // StateIdle/Opening/Open/Closing/Closed
   #diagFault := #fault;
   #diagFaultCode := #faultCode;
END_REGION
END_FUNCTION_BLOCK

// folder: 40. Safety/F-Program

FUNCTION_BLOCK "Main_Safety_RTG1"   // FB1, F_FBD
{ S7_Optimized_Access := 'TRUE' }
BEGIN
END_FUNCTION_BLOCK